LIN {X 0,Y 255.532,Z 417.874,A -85,B 0,C 180,E1 -18352.339,E2 -18352.339} C_VEL
LIN {X 0,Y 254.706,Z 421.868,A -85,B 0,C 180,E1 -18353.296,E2 -18353.296} C_VEL
LIN {X 0,Y 254.484,Z 428.797,A -85,B 0,C 180,E1 -18355.253,E2 -18355.253} C_VEL
LIN {X 0,Y 254.306,Z 433.396,A -85,B 0,C 180,E1 -18356.837,E2 -18356.837} C_VEL
LIN {X 0,Y 254.108,Z 438.832,A -85,B 0,C 180,E1 -18359.213,E2 -18359.213} C_VEL
LIN {X 0,Y 254.235,Z 442.907,A -85,B 0,C 180,E1 -18361.589,E2 -18361.589} C_VEL
LIN {X 0,Y 254.501,Z 444.809,A -85,B 0,C 180,E1 -18363.171,E2 -18363.171} C_VEL
LIN {X 0,Y 254.944,Z 446.181,A -85,B 0,C 180,E1 -18364.749,E2 -18364.749} C_VEL
LIN {X 0,Y 255.447,Z 447.047,A -85,B 0,C 180,E1 -18366.323,E2 -18366.323} C_VEL
LIN {X 0,Y 256.003,Z 447.441,A -85,B 0,C 180,E1 -18367.894,E2 -18367.894} C_VEL
LIN {X 0,Y 256.716,Z 447.298,A -85,B 0,C 180,E1 -18369.459,E2 -18369.459} C_VEL
LIN {X 0,Y 257.985,Z 446.539,A -85,B 0,C 180,E1 -18370.998,E2 -18370.998} C_VEL
LIN {X 0,Y 259.088,Z 445.311,A -85,B 0,C 180,E1 -18372.538,E2 -18372.538} C_VEL
LIN {X 0,Y 261.368,Z 442.495,A -85,B 0,C 180,E1 -18374.805,E2 -18374.805} C_VEL
LIN {X 0,Y 264.023,Z 438.388,A -85,B 0,C 180,E1 -18377.031,E2 -18377.031} C_VEL
LIN {X 0,Y 267.081,Z 432.657,A -85,B 0,C 180,E1 -18379.208,E2 -18379.208} C_VEL
LIN {X 0,Y 270.57,Z 425.346,A -85,B 0,C 180,E1 -18381.329,E2 -18381.329} C_VEL
LIN {X 0,Y 273.754,Z 417.526,A -85,B 0,C 180,E1 -18383.053,E2 -18383.053} C_VEL
LIN {X 0,Y 276.81,Z 408.776,A -85,B 0,C 180,E1 -18384.571,E2 -18384.571} C_VEL
LIN {X 0,Y 280.101,Z 397.834,A -85,B 0,C 180,E1 -18386.05,E2 -18386.05} C_VEL
LIN {X 0,Y 282.427,Z 388.573,A -85,B 0,C 180,E1 -18387.014,E2 -18387.014} C_VEL
LIN {X 0,Y 284.64,Z 377.889,A -85,B 0,C 180,E1 -18387.882,E2 -18387.882} C_VEL
LIN {X 0,Y 286.646,Z 364.758,A -85,B 0,C 180,E1 -18388.634,E2 -18388.634} C_VEL
LIN {X 0,Y 290.224,Z 339.358,A -85,B 0,C 180,E1 -18389.791,E2 -18389.791} C_VEL
LIN {X 0,Y 287.918,Z 334.215,A -85,B 0,C 180,E1 -18391.022,E2 -18391.022} C_VEL
LIN {X 0,Y 285.263,Z 329.062,A -85,B 0,C 180,E1 -18392.583,E2 -18392.583} C_VEL
LIN {X 0,Y 283.342,Z 325.566,A -85,B 0,C 180,E1 -18393.856,E2 -18393.856} C_VEL
LIN {X 0,Y 281.365,Z 322.149,A -85,B 0,C 180,E1 -18395.32,E2 -18395.32} C_VEL
LIN {X 0,Y 278.787,Z 318.232,A -85,B 0,C 180,E1 -18397.663,E2 -18397.663} C_VEL
LIN {X 0,Y 276.577,Z 315.147,A -85,B 0,C 180,E1 -18400.609,E2 -18400.609} C_VEL
LIN {X 0,Y 275.521,Z 314.061,A -85,B 0,C 180,E1 -18403.533,E2 -18403.533} C_VEL
LIN {X 0,Y 275.692,Z 314.436,A -85,B 0,C 180,E1 -18406.695,E2 -18406.695} C_VEL
LIN {X 0,Y 276.651,Z 315.559,A -85,B 0,C 180,E1 -18408.873,E2 -18408.873} C_VEL
LIN {X 0,Y 279.569,Z 320.399,A -85,B 0,C 180,E1 -18412.537,E2 -18412.537} C_VEL
LIN {X 0,Y 282.02,Z 324.321,A -85,B 0,C 180,E1 -18414.58,E2 -18414.58} C_VEL
LIN {X 0,Y 285.054,Z 329.58,A -85,B 0,C 180,E1 -18416.638,E2 -18416.638} C_VEL
LIN {X 0,Y 286.981,Z 333.308,A -85,B 0,C 180,E1 -18417.784,E2 -18417.784} C_VEL
LIN {X 0,Y 287.318,Z 336.449,A -85,B 0,C 180,E1 -18418.229,E2 -18418.229} C_VEL
LIN {X 0,Y 287.621,Z 346.023,A -85,B 0,C 180,E1 -18419.269,E2 -18419.269} C_VEL
LIN {X 0,Y 287.621,Z 359.572,A -85,B 0,C 180,E1 -18420.487,E2 -18420.487} C_VEL
LIN {X 0,Y 285.508,Z 376.187,A -85,B 0,C 180,E1 -18421.308,E2 -18421.308} C_VEL
LIN {X 0,Y 283.222,Z 391.082,A -85,B 0,C 180,E1 -18422.071,E2 -18422.071} C_VEL
LIN {X 0,Y 280.809,Z 401.893,A -85,B 0,C 180,E1 -18422.822,E2 -18422.822} C_VEL
LIN {X 0,Y 277.629,Z 413.56,A -85,B 0,C 180,E1 -18423.906,E2 -18423.906} C_VEL
LIN {X 0,Y 274.246,Z 423.856,A -85,B 0,C 180,E1 -18425.188,E2 -18425.188} C_VEL
LIN {X 0,Y 270.878,Z 433.267,A -85,B 0,C 180,E1 -18426.692,E2 -18426.692} C_VEL
LIN {X 0,Y 267.476,Z 441.522,A -85,B 0,C 180,E1 -18428.416,E2 -18428.416} C_VEL
LIN {X 0,Y 264.494,Z 448.238,A -85,B 0,C 180,E1 -18430.197,E2 -18430.197} C_VEL
LIN {X 0,Y 261.925,Z 453.712,A -85,B 0,C 180,E1 -18432.027,E2 -18432.027} C_VEL
LIN {X 0,Y 259.25,Z 458.894,A -85,B 0,C 180,E1 -18434.271,E2 -18434.271} C_VEL
LIN {X 0,Y 257.239,Z 462.638,A -85,B 0,C 180,E1 -18436.571,E2 -18436.571} C_VEL
LIN {X 0,Y 255.744,Z 465.126,A -85,B 0,C 180,E1 -18438.909,E2 -18438.909} C_VEL
LIN {X 0,Y 255.001,Z 466.213,A -85,B 0,C 180,E1 -18440.481,E2 -18440.481} C_VEL
LIN {X 0,Y 254.485,Z 466.747,A -85,B 0,C 180,E1 -18442.063,E2 -18442.063} C_VEL
LIN {X 0,Y 254.177,Z 466.561,A -85,B 0,C 180,E1 -18444.534,E2 -18444.534} C_VEL
LIN {X 0,Y 254.211,Z 465.734,A -85,B 0,C 180,E1 -18446.433,E2 -18446.433} C_VEL
LIN {X 0,Y 254.165,Z 467.87,A -85,B 0,C 180,E1 -18448.415,E2 -18448.415} C_VEL
LIN {X 0,Y 254.175,Z 468.938,A -85,B 0,C 180,E1 -18450,E2 -18450} C_VEL
LIN {X 0,Y 254.123,Z 469.524,A -85,B 0,C 180,E1 -18451.584,E2 -18451.584} C_VEL
LIN {X 0,Y 254.096,Z 469.648,A -85,B 0,C 180,E1 -18453.171,E2 -18453.171} C_VEL
LIN {X 0,Y 254.098,Z 468.987,A -85,B 0,C 180,E1 -18455.277,E2 -18455.277} C_VEL
LIN {X 0,Y 254.442,Z 466.869,A -85,B 0,C 180,E1 -18457.938,E2 -18457.938} C_VEL
LIN {X 0,Y 255.191,Z 463.773,A -85,B 0,C 180,E1 -18460.312,E2 -18460.312} C_VEL
LIN {X 0,Y 256.366,Z 459.409,A -85,B 0,C 180,E1 -18462.668,E2 -18462.668} C_VEL
LIN {X 0,Y 257.946,Z 453.409,A -85,B 0,C 180,E1 -18465.001,E2 -18465.001} C_VEL
LIN {X 0,Y 259.265,Z 448.471,A -85,B 0,C 180,E1 -18466.536,E2 -18466.536} C_VEL
LIN {X 0,Y 260.845,Z 442.538,A -85,B 0,C 180,E1 -18468.05,E2 -18468.05} C_VEL
LIN {X 0,Y 262.653,Z 435.339,A -85,B 0,C 180,E1 -18469.54,E2 -18469.54} C_VEL
LIN {X 0,Y 264.044,Z 428.911,A -85,B 0,C 180,E1 -18470.651,E2 -18470.651} C_VEL
LIN {X 0,Y 265.617,Z 421.156,A -85,B 0,C 180,E1 -18471.742,E2 -18471.742} C_VEL
LIN {X 0,Y 267.029,Z 413.233,A -85,B 0,C 180,E1 -18472.638,E2 -18472.638} C_VEL
LIN {X 0,Y 268.38,Z 404.327,A -85,B 0,C 180,E1 -18473.419,E2 -18473.419} C_VEL
LIN {X 0,Y 269.583,Z 394.644,A -85,B 0,C 180,E1 -18474.034,E2 -18474.034} C_VEL
LIN {X 0,Y 270.306,Z 385.092,A -85,B 0,C 180,E1 -18474.45,E2 -18474.45} C_VEL
LIN {X 0,Y 271.249,Z 355.127,A -85,B 0,C 180,E1 -18475.292,E2 -18475.292} C_VEL
LIN {X 0,Y 268.624,Z 337.709,A -85,B 0,C 180,E1 -18476.167,E2 -18476.167} C_VEL
LIN {X 0,Y 264.568,Z 317.868,A -85,B 0,C 180,E1 -18477.341,E2 -18477.341} C_VEL
LIN {X 0,Y 262.33,Z 311.832,A -85,B 0,C 180,E1 -18477.854,E2 -18477.854} C_VEL
LIN {X 0,Y 260.483,Z 307.622,A -85,B 0,C 180,E1 -18478.29,E2 -18478.29} C_VEL
LIN {X 0,Y 258.73,Z 299.457,A -85,B 0,C 180,E1 -18481.755,E2 -18481.755} C_VEL
LIN {X 0,Y 256.781,Z 291.051,A -85,B 0,C 180,E1 -18485.563,E2 -18485.563} C_VEL
LIN {X 0,Y 256.133,Z 288.384,A -85,B 0,C 180,E1 -18486.886,E2 -18486.886} C_VEL
LIN {X 0,Y 256.064,Z 288.397,A -85,B 0,C 180,E1 -18491.201,E2 -18491.201} C_VEL
LIN {X 0,Y 256.047,Z 288.404,A -85,B 0,C 180,E1 -18495.532,E2 -18495.532} C_VEL
LIN {X 0,Y 256.018,Z 288.406,A -85,B 0,C 180,E1 -18498.785,E2 -18498.785} C_VEL
LIN {X 0,Y 256.108,Z 288.395,A -85,B 0,C 180,E1 -18502.859,E2 -18502.859} C_VEL
LIN {X 0,Y 256.075,Z 288.398,A -85,B 0,C 180,E1 -18506.704,E2 -18506.704} C_VEL
LIN {X 0,Y 256.064,Z 288.399,A -85,B 0,C 180,E1 -18510.389,E2 -18510.389} C_VEL
LIN {X 0,Y 256.142,Z 288.387,A -85,B 0,C 180,E1 -18514.884,E2 -18514.884} C_VEL
LIN {X 0,Y 256.154,Z 288.377,A -85,B 0,C 180,E1 -18519.099,E2 -18519.099} C_VEL
LIN {X 0,Y 256.264,Z 288.362,A -85,B 0,C 180,E1 -18524.078,E2 -18524.078} C_VEL
LIN {X 0,Y 256.294,Z 288.367,A -85,B 0,C 180,E1 -18527.323,E2 -18527.323} C_VEL
LIN {X 0,Y 256.518,Z 288.339,A -85,B 0,C 180,E1 -18532.122,E2 -18532.122} C_VEL
LIN {X 0,Y 256.487,Z 288.342,A -85,B 0,C 180,E1 -18536.854,E2 -18536.854} C_VEL
LIN {X 0,Y 256.75,Z 288.298,A -85,B 0,C 180,E1 -18539.995,E2 -18539.995} C_VEL
LIN {X 0,Y 256.49,Z 288.343,A -85,B 0,C 180,E1 -18543.136,E2 -18543.136} C_VEL
LIN {X 0,Y 256.492,Z 288.346,A -85,B 0,C 180,E1 -18547.869,E2 -18547.869} C_VEL
LIN {X 0,Y 256.288,Z 288.374,A -85,B 0,C 180,E1 -18552.667,E2 -18552.667} C_VEL
LIN {X 0,Y 256.276,Z 288.365,A -85,B 0,C 180,E1 -18556.297,E2 -18556.297} C_VEL
LIN {X 0,Y 256.148,Z 288.384,A -85,B 0,C 180,E1 -18561.114,E2 -18561.114} C_VEL
LIN {X 0,Y 256.177,Z 288.38,A -85,B 0,C 180,E1 -18565.133,E2 -18565.133} C_VEL
LIN {X 0,Y 256.09,Z 288.397,A -85,B 0,C 180,E1 -18569.596,E2 -18569.596} C_VEL
LIN {X 0,Y 256.052,Z 288.403,A -85,B 0,C 180,E1 -18573.288,E2 -18573.288} C_VEL
LIN {X 0,Y 256.116,Z 288.385,A -85,B 0,C 180,E1 -18577.271,E2 -18577.271} C_VEL
LIN {X 0,Y 256.108,Z 288.387,A -85,B 0,C 180,E1 -18581.184,E2 -18581.184} C_VEL
LIN {X 0,Y 256.148,Z 288.383,A -85,B 0,C 180,E1 -18584.086,E2 -18584.086} C_VEL
LIN {X 0,Y 257.107,Z 291.213,A -85,B 0,C 180,E1 -18584.354,E2 -18584.354} C_VEL
LIN {X 0,Y 258.815,Z 293.87,A -85,B 0,C 180,E1 -18584.707,E2 -18584.707} C_VEL
LIN {X 0,Y 263.773,Z 302.774,A -85,B 0,C 180,E1 -18585.734,E2 -18585.734} C_VEL
LIN {X 0,Y 270.833,Z 318.205,A -85,B 0,C 180,E1 -18587.187,E2 -18587.187} C_VEL
LIN {X 0,Y 272.462,Z 322.528,A -85,B 0,C 180,E1 -18587.532,E2 -18587.532} C_VEL
LIN {X 0,Y 270.884,Z 364.957,A -85,B 0,C 180,E1 -18588.697,E2 -18588.697} C_VEL
LIN {X 0,Y 270.197,Z 375.244,A -85,B 0,C 180,E1 -18589.203,E2 -18589.203} C_VEL
LIN {X 0,Y 268.991,Z 386.83,A -85,B 0,C 180,E1 -18590.078,E2 -18590.078} C_VEL
LIN {X 0,Y 267.757,Z 395.342,A -85,B 0,C 180,E1 -18590.954,E2 -18590.954} C_VEL
LIN {X 0,Y 266.179,Z 404.53,A -85,B 0,C 180,E1 -18592.178,E2 -18592.178} C_VEL
LIN {X 0,Y 264.519,Z 412.588,A -85,B 0,C 180,E1 -18593.525,E2 -18593.525} C_VEL
LIN {X 0,Y 262.892,Z 419.365,A -85,B 0,C 180,E1 -18594.917,E2 -18594.917} C_VEL
LIN {X 0,Y 260.893,Z 427.14,A -85,B 0,C 180,E1 -18596.913,E2 -18596.913} C_VEL
LIN {X 0,Y 259.096,Z 433.249,A -85,B 0,C 180,E1 -18598.978,E2 -18598.978} C_VEL
LIN {X 0,Y 257.954,Z 437.194,A -85,B 0,C 180,E1 -18600.66,E2 -18600.66} C_VEL
LIN {X 0,Y 256.933,Z 440.275,A -85,B 0,C 180,E1 -18602.289,E2 -18602.289} C_VEL
LIN {X 0,Y 256.099,Z 442.685,A -85,B 0,C 180,E1 -18603.955,E2 -18603.955} C_VEL
LIN {X 0,Y 255.374,Z 444.447,A -85,B 0,C 180,E1 -18605.619,E2 -18605.619} C_VEL
LIN {X 0,Y 254.82,Z 445.644,A -85,B 0,C 180,E1 -18607.287,E2 -18607.287} C_VEL
LIN {X 0,Y 254.248,Z 446.491,A -85,B 0,C 180,E1 -18610.004,E2 -18610.004} C_VEL
LIN {X 0,Y 253.968,Z 446.049,A -85,B 0,C 180,E1 -18612.278,E2 -18612.278} C_VEL
LIN {X 0,Y 253.969,Z 445.038,A -85,B 0,C 180,E1 -18613.935,E2 -18613.935} C_VEL
LIN {X 0,Y 254.137,Z 442.565,A -85,B 0,C 180,E1 -18616.405,E2 -18616.405} C_VEL
LIN {X 0,Y 254.518,Z 438.676,A -85,B 0,C 180,E1 -18618.855,E2 -18618.855} C_VEL
LIN {X 0,Y 255.092,Z 433.373,A -85,B 0,C 180,E1 -18621.285,E2 -18621.285} C_VEL
LIN {X 0,Y 255.739,Z 427.604,A -85,B 0,C 180,E1 -18623.318,E2 -18623.318} C_VEL
LIN {X 0,Y 256.559,Z 420.445,A -85,B 0,C 180,E1 -18625.286,E2 -18625.286} C_VEL
LIN {X 0,Y 257.363,Z 413.214,A -85,B 0,C 180,E1 -18626.87,E2 -18626.87} C_VEL
LIN {X 0,Y 258.187,Z 405.508,A -85,B 0,C 180,E1 -18628.245,E2 -18628.245} C_VEL
LIN {X 0,Y 259.028,Z 397.399,A -85,B 0,C 180,E1 -18629.417,E2 -18629.417} C_VEL
LIN {X 0,Y 259.687,Z 389.568,A -85,B 0,C 180,E1 -18630.332,E2 -18630.332} C_VEL
LIN {X 0,Y 260.272,Z 380.968,A -85,B 0,C 180,E1 -18631.124,E2 -18631.124} C_VEL
LIN {X 0,Y 260.767,Z 370.639,A -85,B 0,C 180,E1 -18631.822,E2 -18631.822} C_VEL
LIN {X 0,Y 261.173,Z 358.837,A -85,B 0,C 180,E1 -18632.318,E2 -18632.318} C_VEL
LIN {X 0,Y 262.088,Z 311.721,A -85,B 0,C 180,E1 -18633.604,E2 -18633.604} C_VEL
LIN {X 0,Y 260.06,Z 299.467,A -85,B 0,C 180,E1 -18634.081,E2 -18634.081} C_VEL
LIN {X 0,Y 256.313,Z 288.374,A -85,B 0,C 180,E1 -18634.661,E2 -18634.661} C_VEL
LIN {X 0,Y 256.483,Z 288.346,A -85,B 0,C 180,E1 -18637.875,E2 -18637.875} C_VEL
LIN {X 0,Y 256.23,Z 288.376,A -85,B 0,C 180,E1 -18642.676,E2 -18642.676} C_VEL
LIN {X 0,Y 256.218,Z 288.379,A -85,B 0,C 180,E1 -18646.277,E2 -18646.277} C_VEL
LIN {X 0,Y 256.135,Z 288.391,A -85,B 0,C 180,E1 -18650.898,E2 -18650.898} C_VEL
LIN {X 0,Y 256.105,Z 288.396,A -85,B 0,C 180,E1 -18655.115,E2 -18655.115} C_VEL
LIN {X 0,Y 256.025,Z 288.404,A -85,B 0,C 180,E1 -18659.611,E2 -18659.611} C_VEL
LIN {X 0,Y 256.041,Z 288.4,A -85,B 0,C 180,E1 -18663.297,E2 -18663.297} C_VEL
LIN {X 0,Y 256.093,Z 288.396,A -85,B 0,C 180,E1 -18667.275,E2 -18667.275} C_VEL
LIN {X 0,Y 256.036,Z 288.402,A -85,B 0,C 180,E1 -18672.182,E2 -18672.182} C_VEL
LIN {X 0,Y 256.03,Z 288.403,A -85,B 0,C 180,E1 -18676.675,E2 -18676.675} C_VEL
LIN {X 0,Y 256.055,Z 288.397,A -85,B 0,C 180,E1 -18680.863,E2 -18680.863} C_VEL
LIN {X 0,Y 256.116,Z 288.392,A -85,B 0,C 180,E1 -18682.873,E2 -18682.873} C_VEL
LIN {X 0,Y 256.052,Z 288.398,A -85,B 0,C 180,E1 -18686.712,E2 -18686.712} C_VEL
LIN {X 0,Y 256.043,Z 288.402,A -85,B 0,C 180,E1 -18690.398,E2 -18690.398} C_VEL
LIN {X 0,Y 256.124,Z 288.388,A -85,B 0,C 180,E1 -18694.894,E2 -18694.894} C_VEL
LIN {X 0,Y 256.154,Z 288.375,A -85,B 0,C 180,E1 -18699.11,E2 -18699.11} C_VEL
LIN {X 0,Y 256.386,Z 288.337,A -85,B 0,C 180,E1 -18702.147,E2 -18702.147} C_VEL
LIN {X 0,Y 258.584,Z 308.952,A -85,B 0,C 180,E1 -18703.136,E2 -18703.136} C_VEL
LIN {X 0,Y 257.215,Z 365.235,A -85,B 0,C 180,E1 -18705.72,E2 -18705.72} C_VEL
LIN {X 0,Y 256.873,Z 376.015,A -85,B 0,C 180,E1 -18706.457,E2 -18706.457} C_VEL
LIN {X 0,Y 256.429,Z 387.695,A -85,B 0,C 180,E1 -18707.541,E2 -18707.541} C_VEL
LIN {X 0,Y 255.881,Z 398.365,A -85,B 0,C 180,E1 -18708.881,E2 -18708.881} C_VEL
LIN {X 0,Y 255.407,Z 407.479,A -85,B 0,C 180,E1 -18710.303,E2 -18710.303} C_VEL
LIN {X 0,Y 254.959,Z 416.652,A -85,B 0,C 180,E1 -18712.083,E2 -18712.083} C_VEL
LIN {X 0,Y 254.706,Z 421.868,A -85,B 0,C 180,E1 -18713.296,E2 -18713.296} C_VEL
LIN {X 0,Y 253.879,Z 425.701,A -85,B 0,C 180,E1 -18714.293,E2 -18714.293} C_VEL
LIN {X 0,Y 252.144,Z 429.067,A -85,B 0,C 180,E1 -18715.334,E2 -18715.334} C_VEL
LIN {X 0,Y 247.736,Z 435.645,A -85,B 0,C 180,E1 -18717.981,E2 -18717.981} C_VEL
LIN {X 0,Y 247.036,Z 438.202,A -85,B 0,C 180,E1 -18719.221,E2 -18719.221} C_VEL
LIN {X 0,Y 247.165,Z 442.474,A -85,B 0,C 180,E1 -18721.635,E2 -18721.635} C_VEL
LIN {X 0,Y 247.44,Z 444.59,A -85,B 0,C 180,E1 -18723.262,E2 -18723.262} C_VEL
LIN {X 0,Y 247.875,Z 446.181,A -85,B 0,C 180,E1 -18724.884,E2 -18724.884} C_VEL
LIN {X 0,Y 248.399,Z 447.279,A -85,B 0,C 180,E1 -18726.503,E2 -18726.503} C_VEL
LIN {X 0,Y 248.99,Z 447.808,A -85,B 0,C 180,E1 -18728.118,E2 -18728.118} C_VEL
LIN {X 0,Y 249.748,Z 447.791,A -85,B 0,C 180,E1 -18729.725,E2 -18729.725} C_VEL
LIN {X 0,Y 251.982,Z 446.617,A -85,B 0,C 180,E1 -18732.529,E2 -18732.529} C_VEL
LIN {X 0,Y 253.831,Z 444.809,A -85,B 0,C 180,E1 -18734.434,E2 -18734.434} C_VEL
LIN {X 0,Y 256.432,Z 441.402,A -85,B 0,C 180,E1 -18736.729,E2 -18736.729} C_VEL
LIN {X 0,Y 259.51,Z 436.674,A -85,B 0,C 180,E1 -18738.969,E2 -18738.969} C_VEL
LIN {X 0,Y 262.426,Z 431.601,A -85,B 0,C 180,E1 -18740.789,E2 -18740.789} C_VEL
LIN {X 0,Y 266.277,Z 423.768,A -85,B 0,C 180,E1 -18742.916,E2 -18742.916} C_VEL
LIN {X 0,Y 269.7,Z 415.546,A -85,B 0,C 180,E1 -18744.646,E2 -18744.646} C_VEL
LIN {X 0,Y 273.107,Z 406.397,A -85,B 0,C 180,E1 -18746.152,E2 -18746.152} C_VEL
LIN {X 0,Y 275.839,Z 397.449,A -85,B 0,C 180,E1 -18747.302,E2 -18747.302} C_VEL
LIN {X 0,Y 278.735,Z 386.349,A -85,B 0,C 180,E1 -18748.423,E2 -18748.423} C_VEL
LIN {X 0,Y 281.214,Z 374.18,A -85,B 0,C 180,E1 -18749.324,E2 -18749.324} C_VEL
LIN {X 0,Y 283.64,Z 358.651,A -85,B 0,C 180,E1 -18750.105,E2 -18750.105} C_VEL
LIN {X 0,Y 285.914,Z 342.529,A -85,B 0,C 180,E1 -18750.895,E2 -18750.895} C_VEL
LIN {X 0,Y 282.76,Z 335.677,A -85,B 0,C 180,E1 -18752.844,E2 -18752.844} C_VEL
LIN {X 0,Y 280.376,Z 331.231,A -85,B 0,C 180,E1 -18754.527,E2 -18754.527} C_VEL
LIN {X 0,Y 278.688,Z 328.177,A -85,B 0,C 180,E1 -18755.937,E2 -18755.937} C_VEL
LIN {X 0,Y 276.709,Z 324.937,A -85,B 0,C 180,E1 -18757.898,E2 -18757.898} C_VEL
LIN {X 0,Y 274.619,Z 321.903,A -85,B 0,C 180,E1 -18760.838,E2 -18760.838} C_VEL
LIN {X 0,Y 273.818,Z 320.976,A -85,B 0,C 180,E1 -18763.003,E2 -18763.003} C_VEL
LIN {X 0,Y 273.879,Z 321.279,A -85,B 0,C 180,E1 -18766.582,E2 -18766.582} C_VEL
LIN {X 0,Y 274.736,Z 322.335,A -85,B 0,C 180,E1 -18768.663,E2 -18768.663} C_VEL
LIN {X 0,Y 277.302,Z 326.87,A -85,B 0,C 180,E1 -18772.161,E2 -18772.161} C_VEL
LIN {X 0,Y 279.521,Z 330.618,A -85,B 0,C 180,E1 -18774.154,E2 -18774.154} C_VEL
LIN {X 0,Y 282.209,Z 335.555,A -85,B 0,C 180,E1 -18776.125,E2 -18776.125} C_VEL
LIN {X 0,Y 283.577,Z 338.512,A -85,B 0,C 180,E1 -18777.064,E2 -18777.064} C_VEL
LIN {X 0,Y 283.745,Z 348.629,A -85,B 0,C 180,E1 -18778.198,E2 -18778.198} C_VEL
LIN {X 0,Y 283.486,Z 361.625,A -85,B 0,C 180,E1 -18779.407,E2 -18779.407} C_VEL
LIN {X 0,Y 279.505,Z 388.455,A -85,B 0,C 180,E1 -18780.742,E2 -18780.742} C_VEL
LIN {X 0,Y 276.722,Z 400.474,A -85,B 0,C 180,E1 -18781.562,E2 -18781.562} C_VEL
LIN {X 0,Y 273.346,Z 412.373,A -85,B 0,C 180,E1 -18782.639,E2 -18782.639} C_VEL
LIN {X 0,Y 269.76,Z 422.749,A -85,B 0,C 180,E1 -18783.919,E2 -18783.919} C_VEL
LIN {X 0,Y 266.857,Z 430.22,A -85,B 0,C 180,E1 -18785.078,E2 -18785.078} C_VEL
LIN {X 0,Y 263.126,Z 439.07,A -85,B 0,C 180,E1 -18786.798,E2 -18786.798} C_VEL
LIN {X 0,Y 259.76,Z 446.155,A -85,B 0,C 180,E1 -18788.577,E2 -18788.577} C_VEL
LIN {X 0,Y 257.379,Z 450.864,A -85,B 0,C 180,E1 -18790.042,E2 -18790.042} C_VEL
LIN {X 0,Y 254.317,Z 456.485,A -85,B 0,C 180,E1 -18792.303,E2 -18792.303} C_VEL
LIN {X 0,Y 251.72,Z 460.782,A -85,B 0,C 180,E1 -18794.618,E2 -18794.618} C_VEL
LIN {X 0,Y 249.752,Z 463.822,A -85,B 0,C 180,E1 -18796.99,E2 -18796.99} C_VEL
LIN {X 0,Y 248.765,Z 465.133,A -85,B 0,C 180,E1 -18798.594,E2 -18798.594} C_VEL
LIN {X 0,Y 247.987,Z 465.972,A -85,B 0,C 180,E1 -18800.209,E2 -18800.209} C_VEL
LIN {X 0,Y 247.442,Z 466.357,A -85,B 0,C 180,E1 -18801.835,E2 -18801.835} C_VEL
LIN {X 0,Y 247.184,Z 466.23,A -85,B 0,C 180,E1 -18803.469,E2 -18803.469} C_VEL
LIN {X 0,Y 247.164,Z 464.91,A -85,B 0,C 180,E1 -18806.127,E2 -18806.127} C_VEL
LIN {X 0,Y 247.093,Z 467.393,A -85,B 0,C 180,E1 -18808.37,E2 -18808.37} C_VEL
LIN {X 0,Y 247.099,Z 468.522,A -85,B 0,C 180,E1 -18810,E2 -18810} C_VEL
LIN {X 0,Y 247.051,Z 469.167,A -85,B 0,C 180,E1 -18811.63,E2 -18811.63} C_VEL
LIN {X 0,Y 247.011,Z 469.349,A -85,B 0,C 180,E1 -18813.262,E2 -18813.262} C_VEL
LIN {X 0,Y 247.003,Z 468.88,A -85,B 0,C 180,E1 -18815.181,E2 -18815.181} C_VEL
LIN {X 0,Y 247.402,Z 466.688,A -85,B 0,C 180,E1 -18818.165,E2 -18818.165} C_VEL
LIN {X 0,Y 248.205,Z 463.655,A -85,B 0,C 180,E1 -18820.605,E2 -18820.605} C_VEL
LIN {X 0,Y 249.434,Z 459.378,A -85,B 0,C 180,E1 -18823.026,E2 -18823.026} C_VEL
LIN {X 0,Y 251.104,Z 453.525,A -85,B 0,C 180,E1 -18825.42,E2 -18825.42} C_VEL
LIN {X 0,Y 252.882,Z 447.267,A -85,B 0,C 180,E1 -18827.383,E2 -18827.383} C_VEL
LIN {X 0,Y 254.604,Z 441.165,A -85,B 0,C 180,E1 -18828.925,E2 -18828.925} C_VEL
LIN {X 0,Y 256.237,Z 434.785,A -85,B 0,C 180,E1 -18830.259,E2 -18830.259} C_VEL
LIN {X 0,Y 257.437,Z 429.537,A -85,B 0,C 180,E1 -18831.206,E2 -18831.206} C_VEL
LIN {X 0,Y 259.353,Z 420.498,A -85,B 0,C 180,E1 -18832.505,E2 -18832.505} C_VEL
LIN {X 0,Y 260.848,Z 412.492,A -85,B 0,C 180,E1 -18833.416,E2 -18833.416} C_VEL
LIN {X 0,Y 262.142,Z 404.259,A -85,B 0,C 180,E1 -18834.152,E2 -18834.152} C_VEL
LIN {X 0,Y 263.414,Z 394.577,A -85,B 0,C 180,E1 -18834.78,E2 -18834.78} C_VEL
LIN {X 0,Y 264.136,Z 385.446,A -85,B 0,C 180,E1 -18835.196,E2 -18835.196} C_VEL
LIN {X 0,Y 265.131,Z 356.256,A -85,B 0,C 180,E1 -18836.038,E2 -18836.038} C_VEL
LIN {X 0,Y 263.066,Z 341.866,A -85,B 0,C 180,E1 -18836.774,E2 -18836.774} C_VEL
LIN {X 0,Y 259.448,Z 323.133,A -85,B 0,C 180,E1 -18837.895,E2 -18837.895} C_VEL
LIN {X 0,Y 258.175,Z 318.358,A -85,B 0,C 180,E1 -18838.242,E2 -18838.242} C_VEL
LIN {X 0,Y 254.158,Z 309.74,A -85,B 0,C 180,E1 -18839.145,E2 -18839.145} C_VEL
LIN {X 0,Y 253.208,Z 307.156,A -85,B 0,C 180,E1 -18839.43,E2 -18839.43} C_VEL
LIN {X 0,Y 251.27,Z 298.315,A -85,B 0,C 180,E1 -18843.373,E2 -18843.373} C_VEL
LIN {X 0,Y 249.61,Z 291.26,A -85,B 0,C 180,E1 -18846.749,E2 -18846.749} C_VEL
LIN {X 0,Y 249.043,Z 289.279,A -85,B 0,C 180,E1 -18847.794,E2 -18847.794} C_VEL
LIN {X 0,Y 249.017,Z 289.279,A -85,B 0,C 180,E1 -18850.476,E2 -18850.476} C_VEL
LIN {X 0,Y 248.993,Z 289.277,A -85,B 0,C 180,E1 -18854.881,E2 -18854.881} C_VEL
LIN {X 0,Y 248.993,Z 289.276,A -85,B 0,C 180,E1 -18857.353,E2 -18857.353} C_VEL
LIN {X 0,Y 249.048,Z 289.273,A -85,B 0,C 180,E1 -18862.199,E2 -18862.199} C_VEL
LIN {X 0,Y 249.052,Z 289.267,A -85,B 0,C 180,E1 -18865.636,E2 -18865.636} C_VEL
LIN {X 0,Y 249.011,Z 289.269,A -85,B 0,C 180,E1 -18869.463,E2 -18869.463} C_VEL
LIN {X 0,Y 249.045,Z 289.266,A -85,B 0,C 180,E1 -18873.154,E2 -18873.154} C_VEL
LIN {X 0,Y 249.063,Z 289.272,A -85,B 0,C 180,E1 -18876.726,E2 -18876.726} C_VEL
LIN {X 0,Y 249.096,Z 289.265,A -85,B 0,C 180,E1 -18880.206,E2 -18880.206} C_VEL
LIN {X 0,Y 249.201,Z 289.242,A -85,B 0,C 180,E1 -18883.614,E2 -18883.614} C_VEL
LIN {X 0,Y 249.247,Z 289.232,A -85,B 0,C 180,E1 -18888.611,E2 -18888.611} C_VEL
LIN {X 0,Y 249.458,Z 289.22,A -85,B 0,C 180,E1 -18891.897,E2 -18891.897} C_VEL
LIN {X 0,Y 249.285,Z 289.229,A -85,B 0,C 180,E1 -18895.143,E2 -18895.143} C_VEL
LIN {X 0,Y 249.672,Z 289.187,A -85,B 0,C 180,E1 -18898.382,E2 -18898.382} C_VEL
LIN {X 0,Y 249.672,Z 289.188,A -85,B 0,C 180,E1 -18901.608,E2 -18901.608} C_VEL
LIN {X 0,Y 249.427,Z 289.217,A -85,B 0,C 180,E1 -18906.58,E2 -18906.58} C_VEL
LIN {X 0,Y 249.339,Z 289.229,A -85,B 0,C 180,E1 -18909.731,E2 -18909.731} C_VEL
LIN {X 0,Y 249.199,Z 289.249,A -85,B 0,C 180,E1 -18914.698,E2 -18914.698} C_VEL
LIN {X 0,Y 249.132,Z 289.265,A -85,B 0,C 180,E1 -18918.072,E2 -18918.072} C_VEL
LIN {X 0,Y 249.078,Z 289.267,A -85,B 0,C 180,E1 -18921.513,E2 -18921.513} C_VEL
LIN {X 0,Y 249.119,Z 289.262,A -85,B 0,C 180,E1 -18925.477,E2 -18925.477} C_VEL
LIN {X 0,Y 249.06,Z 289.269,A -85,B 0,C 180,E1 -18928.984,E2 -18928.984} C_VEL
LIN {X 0,Y 249.015,Z 289.276,A -85,B 0,C 180,E1 -18932.421,E2 -18932.421} C_VEL
LIN {X 0,Y 249.043,Z 289.258,A -85,B 0,C 180,E1 -18936.335,E2 -18936.335} C_VEL
LIN {X 0,Y 249.064,Z 289.261,A -85,B 0,C 180,E1 -18940.458,E2 -18940.458} C_VEL
LIN {X 0,Y 249.073,Z 289.27,A -85,B 0,C 180,E1 -18942.986,E2 -18942.986} C_VEL
LIN {X 0,Y 250.053,Z 292.07,A -85,B 0,C 180,E1 -18943.253,E2 -18943.253} C_VEL
LIN {X 0,Y 251.663,Z 294.475,A -85,B 0,C 180,E1 -18943.602,E2 -18943.602} C_VEL
LIN {X 0,Y 257.999,Z 305.545,A -85,B 0,C 180,E1 -18944.976,E2 -18944.976} C_VEL
LIN {X 0,Y 263.869,Z 318.195,A -85,B 0,C 180,E1 -18946.249,E2 -18946.249} C_VEL
LIN {X 0,Y 266.364,Z 324.215,A -85,B 0,C 180,E1 -18946.783,E2 -18946.783} C_VEL
LIN {X 0,Y 264.785,Z 365.07,A -85,B 0,C 180,E1 -18947.927,E2 -18947.927} C_VEL
LIN {X 0,Y 264.146,Z 374.652,A -85,B 0,C 180,E1 -18948.401,E2 -18948.401} C_VEL
LIN {X 0,Y 262.965,Z 385.914,A -85,B 0,C 180,E1 -18949.223,E2 -18949.223} C_VEL
LIN {X 0,Y 261.374,Z 396.3,A -85,B 0,C 180,E1 -18950.312,E2 -18950.312} C_VEL
LIN {X 0,Y 260.044,Z 403.809,A -85,B 0,C 180,E1 -18951.32,E2 -18951.32} C_VEL
LIN {X 0,Y 258.647,Z 410.534,A -85,B 0,C 180,E1 -18952.408,E2 -18952.408} C_VEL
LIN {X 0,Y 256.765,Z 418.256,A -85,B 0,C 180,E1 -18953.951,E2 -18953.951} C_VEL
LIN {X 0,Y 255.192,Z 424.21,A -85,B 0,C 180,E1 -18955.412,E2 -18955.412} C_VEL
LIN {X 0,Y 253.78,Z 429.083,A -85,B 0,C 180,E1 -18956.843,E2 -18956.843} C_VEL
LIN {X 0,Y 252.314,Z 433.775,A -85,B 0,C 180,E1 -18958.516,E2 -18958.516} C_VEL
LIN {X 0,Y 251.154,Z 437.513,A -85,B 0,C 180,E1 -18960.151,E2 -18960.151} C_VEL
LIN {X 0,Y 249.802,Z 441.336,A -85,B 0,C 180,E1 -18962.341,E2 -18962.341} C_VEL
LIN {X 0,Y 248.582,Z 444.438,A -85,B 0,C 180,E1 -18964.907,E2 -18964.907} C_VEL
LIN {X 0,Y 247.918,Z 445.776,A -85,B 0,C 180,E1 -18966.617,E2 -18966.617} C_VEL
LIN {X 0,Y 247.465,Z 446.573,A -85,B 0,C 180,E1 -18968.334,E2 -18968.334} C_VEL
LIN {X 0,Y 247.153,Z 446.834,A -85,B 0,C 180,E1 -18970.048,E2 -18970.048} C_VEL
LIN {X 0,Y 246.929,Z 446.483,A -85,B 0,C 180,E1 -18971.755,E2 -18971.755} C_VEL
LIN {X 0,Y 246.855,Z 445.582,A -85,B 0,C 180,E1 -18973.459,E2 -18973.459} C_VEL
LIN {X 0,Y 246.929,Z 443.947,A -85,B 0,C 180,E1 -18975.368,E2 -18975.368} C_VEL
LIN {X 0,Y 247.236,Z 440.989,A -85,B 0,C 180,E1 -18977.691,E2 -18977.691} C_VEL
LIN {X 0,Y 247.725,Z 436.459,A -85,B 0,C 180,E1 -18980.2,E2 -18980.2} C_VEL
LIN {X 0,Y 248.28,Z 431.771,A -85,B 0,C 180,E1 -18982.141,E2 -18982.141} C_VEL
LIN {X 0,Y 248.792,Z 426.457,A -85,B 0,C 180,E1 -18983.919,E2 -18983.919} C_VEL
LIN {X 0,Y 249.554,Z 420.461,A -85,B 0,C 180,E1 -18985.559,E2 -18985.559} C_VEL
LIN {X 0,Y 250.394,Z 413.168,A -85,B 0,C 180,E1 -18987.185,E2 -18987.185} C_VEL
LIN {X 0,Y 251.27,Z 405.38,A -85,B 0,C 180,E1 -18988.598,E2 -18988.598} C_VEL
LIN {X 0,Y 252.126,Z 397.179,A -85,B 0,C 180,E1 -18989.801,E2 -18989.801} C_VEL
LIN {X 0,Y 252.8,Z 389.539,A -85,B 0,C 180,E1 -18990.705,E2 -18990.705} C_VEL
LIN {X 0,Y 253.455,Z 379.956,A -85,B 0,C 180,E1 -18991.589,E2 -18991.589} C_VEL
LIN {X 0,Y 254.001,Z 369.105,A -85,B 0,C 180,E1 -18992.306,E2 -18992.306} C_VEL
LIN {X 0,Y 254.389,Z 354.396,A -85,B 0,C 180,E1 -18992.841,E2 -18992.841} C_VEL
LIN {X 0,Y 255.313,Z 312.699,A -85,B 0,C 180,E1 -18994.001,E2 -18994.001} C_VEL
LIN {X 0,Y 253.275,Z 300.812,A -85,B 0,C 180,E1 -18994.485,E2 -18994.485} C_VEL
LIN {X 0,Y 249.307,Z 289.354,A -85,B 0,C 180,E1 -18995.099,E2 -18995.099} C_VEL
LIN {X 0,Y 249.423,Z 289.225,A -85,B 0,C 180,E1 -18998.099,E2 -18998.099} C_VEL
LIN {X 0,Y 249.163,Z 289.258,A -85,B 0,C 180,E1 -19003.042,E2 -19003.042} C_VEL
LIN {X 0,Y 249.166,Z 289.257,A -85,B 0,C 180,E1 -19006.488,E2 -19006.488} C_VEL
LIN {X 0,Y 249.066,Z 289.276,A -85,B 0,C 180,E1 -19011.401,E2 -19011.401} C_VEL
LIN {X 0,Y 249.058,Z 289.275,A -85,B 0,C 180,E1 -19015.463,E2 -19015.463} C_VEL
LIN {X 0,Y 249.008,Z 289.279,A -85,B 0,C 180,E1 -19018.976,E2 -19018.976} C_VEL
LIN {X 0,Y 249.002,Z 289.274,A -85,B 0,C 180,E1 -19022.43,E2 -19022.43} C_VEL
LIN {X 0,Y 248.989,Z 289.279,A -85,B 0,C 180,E1 -19026.353,E2 -19026.353} C_VEL
LIN {X 0,Y 248.962,Z 289.283,A -85,B 0,C 180,E1 -19030.487,E2 -19030.487} C_VEL
LIN {X 0,Y 248.963,Z 289.281,A -85,B 0,C 180,E1 -19034.889,E2 -19034.889} C_VEL
LIN {X 0,Y 248.991,Z 289.281,A -85,B 0,C 180,E1 -19037.366,E2 -19037.366} C_VEL
LIN {X 0,Y 249.01,Z 289.278,A -85,B 0,C 180,E1 -19041.625,E2 -19041.625} C_VEL
LIN {X 0,Y 249.03,Z 289.278,A -85,B 0,C 180,E1 -19045.645,E2 -19045.645} C_VEL
LIN {X 0,Y 248.99,Z 289.28,A -85,B 0,C 180,E1 -19049.472,E2 -19049.472} C_VEL
LIN {X 0,Y 249.025,Z 289.275,A -85,B 0,C 180,E1 -19053.164,E2 -19053.164} C_VEL
LIN {X 0,Y 249.047,Z 289.265,A -85,B 0,C 180,E1 -19056.736,E2 -19056.736} C_VEL
LIN {X 0,Y 249.345,Z 289.214,A -85,B 0,C 180,E1 -19062.131,E2 -19062.131} C_VEL
LIN {X 0,Y 251.494,Z 310.031,A -85,B 0,C 180,E1 -19063.145,E2 -19063.145} C_VEL
LIN {X 0,Y 250.111,Z 365.964,A -85,B 0,C 180,E1 -19065.824,E2 -19065.824} C_VEL
LIN {X 0,Y 249.729,Z 376.583,A -85,B 0,C 180,E1 -19066.581,E2 -19066.581} C_VEL
LIN {X 0,Y 249.369,Z 387.298,A -85,B 0,C 180,E1 -19067.596,E2 -19067.596} C_VEL
LIN {X 0,Y 248.785,Z 398.415,A -85,B 0,C 180,E1 -19069.013,E2 -19069.013} C_VEL
LIN {X 0,Y 248.326,Z 407.345,A -85,B 0,C 180,E1 -19070.435,E2 -19070.435} C_VEL
LIN {X 0,Y 247.874,Z 416.601,A -85,B 0,C 180,E1 -19072.266,E2 -19072.266} C_VEL
LIN {X 0,Y 247.525,Z 423.237,A -85,B 0,C 180,E1 -19073.903,E2 -19073.903} C_VEL
LIN {X 0,Y 247.409,Z 429.995,A -85,B 0,C 180,E1 -19075.933,E2 -19075.933} C_VEL
LIN {X 0,Y 247.104,Z 435.434,A -85,B 0,C 180,E1 -19077.968,E2 -19077.968} C_VEL
LIN {X 0,Y 247.036,Z 438.202,A -85,B 0,C 180,E1 -19079.221,E2 -19079.221} C_VEL
LIN {X 0,Y 246.403,Z 440.606,A -85,B 0,C 180,E1 -19080.475,E2 -19080.475} C_VEL
LIN {X 0,Y 243.774,Z 443.625,A -85,B 0,C 180,E1 -19082.592,E2 -19082.592} C_VEL
LIN {X 0,Y 241.73,Z 445.491,A -85,B 0,C 180,E1 -19084.357,E2 -19084.357} C_VEL
LIN {X 0,Y 241.095,Z 446.672,A -85,B 0,C 180,E1 -19085.732,E2 -19085.732} C_VEL
LIN {X 0,Y 241.171,Z 446.982,A -85,B 0,C 180,E1 -19086.195,E2 -19086.195} C_VEL
LIN {X 0,Y 241.964,Z 448.044,A -85,B 0,C 180,E1 -19088.356,E2 -19088.356} C_VEL
LIN {X 0,Y 242.776,Z 448.285,A -85,B 0,C 180,E1 -19090.008,E2 -19090.008} C_VEL
LIN {X 0,Y 244.143,Z 448.032,A -85,B 0,C 180,E1 -19091.63,E2 -19091.63} C_VEL
LIN {X 0,Y 245.387,Z 447.256,A -85,B 0,C 180,E1 -19093.25,E2 -19093.25} C_VEL
LIN {X 0,Y 247.046,Z 445.874,A -85,B 0,C 180,E1 -19094.84,E2 -19094.84} C_VEL
LIN {X 0,Y 249.802,Z 442.956,A -85,B 0,C 180,E1 -19097.187,E2 -19097.187} C_VEL
LIN {X 0,Y 253.046,Z 438.615,A -85,B 0,C 180,E1 -19099.473,E2 -19099.473} C_VEL
LIN {X 0,Y 256.052,Z 433.86,A -85,B 0,C 180,E1 -19101.331,E2 -19101.331} C_VEL
LIN {X 0,Y 259.38,Z 427.992,A -85,B 0,C 180,E1 -19103.139,E2 -19103.139} C_VEL
LIN {X 0,Y 262.98,Z 420.779,A -85,B 0,C 180,E1 -19104.897,E2 -19104.897} C_VEL
LIN {X 0,Y 266.815,Z 411.613,A -85,B 0,C 180,E1 -19106.606,E2 -19106.606} C_VEL
LIN {X 0,Y 270.099,Z 402.671,A -85,B 0,C 180,E1 -19107.932,E2 -19107.932} C_VEL
LIN {X 0,Y 273.568,Z 391.333,A -85,B 0,C 180,E1 -19109.221,E2 -19109.221} C_VEL
LIN {X 0,Y 276.014,Z 381.224,A -85,B 0,C 180,E1 -19110.09,E2 -19110.09} C_VEL
LIN {X 0,Y 278.297,Z 369.687,A -85,B 0,C 180,E1 -19110.829,E2 -19110.829} C_VEL
LIN {X 0,Y 281.944,Z 346.313,A -85,B 0,C 180,E1 -19111.977,E2 -19111.977} C_VEL
LIN {X 0,Y 279.589,Z 341.037,A -85,B 0,C 180,E1 -19113.61,E2 -19113.61} C_VEL
LIN {X 0,Y 277.823,Z 337.512,A -85,B 0,C 180,E1 -19114.961,E2 -19114.961} C_VEL
LIN {X 0,Y 276.141,Z 334.34,A -85,B 0,C 180,E1 -19116.468,E2 -19116.468} C_VEL
LIN {X 0,Y 274.49,Z 331.478,A -85,B 0,C 180,E1 -19118.277,E2 -19118.277} C_VEL
LIN {X 0,Y 272.658,Z 328.588,A -85,B 0,C 180,E1 -19121.209,E2 -19121.209} C_VEL
LIN {X 0,Y 271.925,Z 327.798,A -85,B 0,C 180,E1 -19123.641,E2 -19123.641} C_VEL
LIN {X 0,Y 272.215,Z 328.277,A -85,B 0,C 180,E1 -19127.072,E2 -19127.072} C_VEL
LIN {X 0,Y 272.865,Z 329.27,A -85,B 0,C 180,E1 -19128.591,E2 -19128.591} C_VEL
LIN {X 0,Y 275.214,Z 333.651,A -85,B 0,C 180,E1 -19131.969,E2 -19131.969} C_VEL
LIN {X 0,Y 277.012,Z 336.938,A -85,B 0,C 180,E1 -19133.719,E2 -19133.719} C_VEL
LIN {X 0,Y 279.476,Z 341.763,A -85,B 0,C 180,E1 -19135.68,E2 -19135.68} C_VEL
LIN {X 0,Y 280.154,Z 343.254,A -85,B 0,C 180,E1 -19136.168,E2 -19136.168} C_VEL
LIN {X 0,Y 279.997,Z 352.566,A -85,B 0,C 180,E1 -19137.227,E2 -19137.227} C_VEL
LIN {X 0,Y 279.599,Z 363.72,A -85,B 0,C 180,E1 -19138.268,E2 -19138.268} C_VEL
LIN {X 0,Y 275.744,Z 387.327,A -85,B 0,C 180,E1 -19139.459,E2 -19139.459} C_VEL
LIN {X 0,Y 272.823,Z 399.55,A -85,B 0,C 180,E1 -19140.272,E2 -19140.272} C_VEL
LIN {X 0,Y 269.778,Z 409.853,A -85,B 0,C 180,E1 -19141.187,E2 -19141.187} C_VEL
LIN {X 0,Y 265.883,Z 420.689,A -85,B 0,C 180,E1 -19142.446,E2 -19142.446} C_VEL
LIN {X 0,Y 262.364,Z 429.31,A -85,B 0,C 180,E1 -19143.769,E2 -19143.769} C_VEL
LIN {X 0,Y 259.059,Z 436.575,A -85,B 0,C 180,E1 -19145.134,E2 -19145.134} C_VEL
LIN {X 0,Y 255.354,Z 444.058,A -85,B 0,C 180,E1 -19146.908,E2 -19146.908} C_VEL
LIN {X 0,Y 251.416,Z 451.117,A -85,B 0,C 180,E1 -19149.12,E2 -19149.12} C_VEL
LIN {X 0,Y 248.625,Z 455.786,A -85,B 0,C 180,E1 -19151.029,E2 -19151.029} C_VEL
LIN {X 0,Y 245.663,Z 460.104,A -85,B 0,C 180,E1 -19153.376,E2 -19153.376} C_VEL
LIN {X 0,Y 244.158,Z 462.279,A -85,B 0,C 180,E1 -19154.985,E2 -19154.985} C_VEL
LIN {X 0,Y 242.841,Z 463.97,A -85,B 0,C 180,E1 -19156.613,E2 -19156.613} C_VEL
LIN {X 0,Y 241.802,Z 465.144,A -85,B 0,C 180,E1 -19158.261,E2 -19158.261} C_VEL
LIN {X 0,Y 240.989,Z 465.738,A -85,B 0,C 180,E1 -19159.922,E2 -19159.922} C_VEL
LIN {X 0,Y 240.418,Z 465.868,A -85,B 0,C 180,E1 -19161.595,E2 -19161.595} C_VEL
LIN {X 0,Y 240.107,Z 465.044,A -85,B 0,C 180,E1 -19164.412,E2 -19164.412} C_VEL
LIN {X 0,Y 240.133,Z 464.136,A -85,B 0,C 180,E1 -19165.85,E2 -19165.85} C_VEL
LIN {X 0,Y 240.023,Z 466.917,A -85,B 0,C 180,E1 -19168.322,E2 -19168.322} C_VEL
LIN {X 0,Y 240.025,Z 468.105,A -85,B 0,C 180,E1 -19170,E2 -19170} C_VEL
LIN {X 0,Y 239.979,Z 468.809,A -85,B 0,C 180,E1 -19171.678,E2 -19171.678} C_VEL
LIN {X 0,Y 239.927,Z 469.039,A -85,B 0,C 180,E1 -19173.358,E2 -19173.358} C_VEL
LIN {X 0,Y 239.925,Z 468.661,A -85,B 0,C 180,E1 -19175.126,E2 -19175.126} C_VEL
LIN {X 0,Y 240.046,Z 467.827,A -85,B 0,C 180,E1 -19176.725,E2 -19176.725} C_VEL
LIN {X 0,Y 240.358,Z 466.514,A -85,B 0,C 180,E1 -19178.406,E2 -19178.406} C_VEL
LIN {X 0,Y 241.202,Z 463.551,A -85,B 0,C 180,E1 -19180.917,E2 -19180.917} C_VEL
LIN {X 0,Y 242.026,Z 460.878,A -85,B 0,C 180,E1 -19182.579,E2 -19182.579} C_VEL
LIN {X 0,Y 243.601,Z 455.682,A -85,B 0,C 180,E1 -19185.049,E2 -19185.049} C_VEL
LIN {X 0,Y 245.722,Z 448.893,A -85,B 0,C 180,E1 -19187.476,E2 -19187.476} C_VEL
LIN {X 0,Y 247.925,Z 441.497,A -85,B 0,C 180,E1 -19189.456,E2 -19189.456} C_VEL
LIN {X 0,Y 249.816,Z 434.234,A -85,B 0,C 180,E1 -19191.02,E2 -19191.02} C_VEL
LIN {X 0,Y 251.473,Z 427.707,A -85,B 0,C 180,E1 -19192.166,E2 -19192.166} C_VEL
LIN {X 0,Y 253.16,Z 419.837,A -85,B 0,C 180,E1 -19193.303,E2 -19193.303} C_VEL
LIN {X 0,Y 254.716,Z 411.75,A -85,B 0,C 180,E1 -19194.231,E2 -19194.231} C_VEL
LIN {X 0,Y 256.143,Z 403.134,A -85,B 0,C 180,E1 -19194.995,E2 -19194.995} C_VEL
LIN {X 0,Y 257.33,Z 393.916,A -85,B 0,C 180,E1 -19195.598,E2 -19195.598} C_VEL
LIN {X 0,Y 258.11,Z 384.471,A -85,B 0,C 180,E1 -19196.023,E2 -19196.023} C_VEL
LIN {X 0,Y 259.09,Z 357.343,A -85,B 0,C 180,E1 -19196.817,E2 -19196.817} C_VEL
LIN {X 0,Y 256.624,Z 340.416,A -85,B 0,C 180,E1 -19197.73,E2 -19197.73} C_VEL
LIN {X 0,Y 253.083,Z 322.491,A -85,B 0,C 180,E1 -19198.873,E2 -19198.873} C_VEL
LIN {X 0,Y 247.58,Z 310.545,A -85,B 0,C 180,E1 -19200.176,E2 -19200.176} C_VEL
LIN {X 0,Y 245.935,Z 306.775,A -85,B 0,C 180,E1 -19200.618,E2 -19200.618} C_VEL
LIN {X 0,Y 244.007,Z 298.078,A -85,B 0,C 180,E1 -19204.702,E2 -19204.702} C_VEL
LIN {X 0,Y 242.613,Z 292.586,A -85,B 0,C 180,E1 -19207.468,E2 -19207.468} C_VEL
LIN {X 0,Y 241.972,Z 290.154,A -85,B 0,C 180,E1 -19208.776,E2 -19208.776} C_VEL
LIN {X 0,Y 241.935,Z 290.159,A -85,B 0,C 180,E1 -19213.423,E2 -19213.423} C_VEL
LIN {X 0,Y 241.918,Z 290.158,A -85,B 0,C 180,E1 -19218.068,E2 -19218.068} C_VEL
LIN {X 0,Y 241.989,Z 290.154,A -85,B 0,C 180,E1 -19222.413,E2 -19222.413} C_VEL
LIN {X 0,Y 241.988,Z 290.153,A -85,B 0,C 180,E1 -19226.504,E2 -19226.504} C_VEL
LIN {X 0,Y 241.986,Z 290.153,A -85,B 0,C 180,E1 -19230.608,E2 -19230.608} C_VEL
LIN {X 0,Y 242.04,Z 290.138,A -85,B 0,C 180,E1 -19234.175,E2 -19234.175} C_VEL
LIN {X 0,Y 242.029,Z 290.136,A -85,B 0,C 180,E1 -19238.311,E2 -19238.311} C_VEL
LIN {X 0,Y 242.133,Z 290.123,A -85,B 0,C 180,E1 -19243.302,E2 -19243.302} C_VEL
LIN {X 0,Y 242.183,Z 290.114,A -85,B 0,C 180,E1 -19248.275,E2 -19248.275} C_VEL
LIN {X 0,Y 242.404,Z 290.097,A -85,B 0,C 180,E1 -19251.66,E2 -19251.66} C_VEL
LIN {X 0,Y 242.425,Z 290.087,A -85,B 0,C 180,E1 -19253.336,E2 -19253.336} C_VEL
LIN {X 0,Y 242.632,Z 290.064,A -85,B 0,C 180,E1 -19258.335,E2 -19258.335} C_VEL
LIN {X 0,Y 242.633,Z 290.065,A -85,B 0,C 180,E1 -19261.654,E2 -19261.654} C_VEL
LIN {X 0,Y 242.404,Z 290.093,A -85,B 0,C 180,E1 -19266.654,E2 -19266.654} C_VEL
LIN {X 0,Y 242.263,Z 290.108,A -85,B 0,C 180,E1 -19270.018,E2 -19270.018} C_VEL
LIN {X 0,Y 242.16,Z 290.123,A -85,B 0,C 180,E1 -19275.135,E2 -19275.135} C_VEL
LIN {X 0,Y 242.065,Z 290.143,A -85,B 0,C 180,E1 -19278.618,E2 -19278.618} C_VEL
LIN {X 0,Y 242.003,Z 290.151,A -85,B 0,C 180,E1 -19282.174,E2 -19282.174} C_VEL
LIN {X 0,Y 242.055,Z 290.143,A -85,B 0,C 180,E1 -19285.832,E2 -19285.832} C_VEL
LIN {X 0,Y 241.994,Z 290.153,A -85,B 0,C 180,E1 -19289.578,E2 -19289.578} C_VEL
LIN {X 0,Y 241.966,Z 290.158,A -85,B 0,C 180,E1 -19293.487,E2 -19293.487} C_VEL
LIN {X 0,Y 241.989,Z 290.148,A -85,B 0,C 180,E1 -19297.574,E2 -19297.574} C_VEL
LIN {X 0,Y 242.005,Z 290.148,A -85,B 0,C 180,E1 -19301.764,E2 -19301.764} C_VEL
LIN {X 0,Y 243.018,Z 293.016,A -85,B 0,C 180,E1 -19302.068,E2 -19302.068} C_VEL
LIN {X 0,Y 244.646,Z 295.216,A -85,B 0,C 180,E1 -19302.44,E2 -19302.44} C_VEL
LIN {X 0,Y 252.319,Z 308.399,A -85,B 0,C 180,E1 -19304.194,E2 -19304.194} C_VEL
LIN {X 0,Y 258.347,Z 321.385,A -85,B 0,C 180,E1 -19305.56,E2 -19305.56} C_VEL
LIN {X 0,Y 260.297,Z 326.197,A -85,B 0,C 180,E1 -19306.004,E2 -19306.004} C_VEL
LIN {X 0,Y 258.75,Z 364.976,A -85,B 0,C 180,E1 -19307.113,E2 -19307.113} C_VEL
LIN {X 0,Y 258.097,Z 374.179,A -85,B 0,C 180,E1 -19307.562,E2 -19307.562} C_VEL
LIN {X 0,Y 257.142,Z 383.5,A -85,B 0,C 180,E1 -19308.226,E2 -19308.226} C_VEL
LIN {X 0,Y 255.651,Z 394.003,A -85,B 0,C 180,E1 -19309.24,E2 -19309.24} C_VEL
LIN {X 0,Y 253.677,Z 404.516,A -85,B 0,C 180,E1 -19310.646,E2 -19310.646} C_VEL
LIN {X 0,Y 252.133,Z 411.451,A -85,B 0,C 180,E1 -19311.808,E2 -19311.808} C_VEL
LIN {X 0,Y 250.211,Z 418.938,A -85,B 0,C 180,E1 -19313.354,E2 -19313.354} C_VEL
LIN {X 0,Y 248.429,Z 425.298,A -85,B 0,C 180,E1 -19314.981,E2 -19314.981} C_VEL
LIN {X 0,Y 246.698,Z 430.888,A -85,B 0,C 180,E1 -19316.743,E2 -19316.743} C_VEL
LIN {X 0,Y 245.227,Z 435.306,A -85,B 0,C 180,E1 -19318.465,E2 -19318.465} C_VEL
LIN {X 0,Y 243.69,Z 439.697,A -85,B 0,C 180,E1 -19320.641,E2 -19320.641} C_VEL
LIN {X 0,Y 242.196,Z 443.561,A -85,B 0,C 180,E1 -19323.271,E2 -19323.271} C_VEL
LIN {X 0,Y 241.081,Z 445.912,A -85,B 0,C 180,E1 -19325.913,E2 -19325.913} C_VEL
LIN {X 0,Y 240.547,Z 446.835,A -85,B 0,C 180,E1 -19327.678,E2 -19327.678} C_VEL
LIN {X 0,Y 240.16,Z 447.144,A -85,B 0,C 180,E1 -19329.442,E2 -19329.442} C_VEL
LIN {X 0,Y 239.89,Z 446.888,A -85,B 0,C 180,E1 -19331.2,E2 -19331.2} C_VEL
LIN {X 0,Y 239.76,Z 446.121,A -85,B 0,C 180,E1 -19332.955,E2 -19332.955} C_VEL
LIN {X 0,Y 239.829,Z 444.332,A -85,B 0,C 180,E1 -19335.219,E2 -19335.219} C_VEL
LIN {X 0,Y 240.068,Z 441.804,A -85,B 0,C 180,E1 -19337.317,E2 -19337.317} C_VEL
LIN {X 0,Y 240.362,Z 439.04,A -85,B 0,C 180,E1 -19339.044,E2 -19339.044} C_VEL
LIN {X 0,Y 240.744,Z 435.629,A -85,B 0,C 180,E1 -19340.761,E2 -19340.761} C_VEL
LIN {X 0,Y 241.369,Z 430.709,A -85,B 0,C 180,E1 -19342.741,E2 -19342.741} C_VEL
LIN {X 0,Y 241.951,Z 425.052,A -85,B 0,C 180,E1 -19344.583,E2 -19344.583} C_VEL
LIN {X 0,Y 242.765,Z 418.716,A -85,B 0,C 180,E1 -19346.266,E2 -19346.266} C_VEL
LIN {X 0,Y 243.559,Z 412.053,A -85,B 0,C 180,E1 -19347.726,E2 -19347.726} C_VEL
LIN {X 0,Y 244.528,Z 403.96,A -85,B 0,C 180,E1 -19349.177,E2 -19349.177} C_VEL
LIN {X 0,Y 245.619,Z 393.319,A -85,B 0,C 180,E1 -19350.677,E2 -19350.677} C_VEL
LIN {X 0,Y 246.367,Z 383.047,A -85,B 0,C 180,E1 -19351.732,E2 -19351.732} C_VEL
LIN {X 0,Y 246.952,Z 373.384,A -85,B 0,C 180,E1 -19352.456,E2 -19352.456} C_VEL
LIN {X 0,Y 247.307,Z 363.974,A -85,B 0,C 180,E1 -19352.938,E2 -19352.938} C_VEL
LIN {X 0,Y 248.493,Z 313.52,A -85,B 0,C 180,E1 -19354.426,E2 -19354.426} C_VEL
LIN {X 0,Y 246.7,Z 303.05,A -85,B 0,C 180,E1 -19354.865,E2 -19354.865} C_VEL
LIN {X 0,Y 242.286,Z 290.118,A -85,B 0,C 180,E1 -19355.58,E2 -19355.58} C_VEL
LIN {X 0,Y 242.369,Z 290.104,A -85,B 0,C 180,E1 -19358.337,E2 -19358.337} C_VEL
LIN {X 0,Y 242.111,Z 290.14,A -85,B 0,C 180,E1 -19363.428,E2 -19363.428} C_VEL
LIN {X 0,Y 242.114,Z 290.137,A -85,B 0,C 180,E1 -19366.875,E2 -19366.875} C_VEL
LIN {X 0,Y 241.998,Z 290.154,A -85,B 0,C 180,E1 -19371.689,E2 -19371.689} C_VEL
LIN {X 0,Y 242.006,Z 290.152,A -85,B 0,C 180,E1 -19375.824,E2 -19375.824} C_VEL
LIN {X 0,Y 241.942,Z 290.158,A -85,B 0,C 180,E1 -19379.593,E2 -19379.593} C_VEL
LIN {X 0,Y 241.954,Z 290.155,A -85,B 0,C 180,E1 -19383.497,E2 -19383.497} C_VEL
LIN {X 0,Y 241.96,Z 290.157,A -85,B 0,C 180,E1 -19387.588,E2 -19387.588} C_VEL
LIN {X 0,Y 241.901,Z 290.164,A -85,B 0,C 180,E1 -19391.931,E2 -19391.931} C_VEL
LIN {X 0,Y 241.906,Z 290.162,A -85,B 0,C 180,E1 -19396.579,E2 -19396.579} C_VEL
LIN {X 0,Y 241.94,Z 290.156,A -85,B 0,C 180,E1 -19400.286,E2 -19400.286} C_VEL
LIN {X 0,Y 241.974,Z 290.154,A -85,B 0,C 180,E1 -19404.495,E2 -19404.495} C_VEL
LIN {X 0,Y 241.94,Z 290.157,A -85,B 0,C 180,E1 -19408.482,E2 -19408.482} C_VEL
LIN {X 0,Y 241.957,Z 290.157,A -85,B 0,C 180,E1 -19412.314,E2 -19412.314} C_VEL
LIN {X 0,Y 242.017,Z 290.145,A -85,B 0,C 180,E1 -19416.019,E2 -19416.019} C_VEL
LIN {X 0,Y 242.201,Z 290.107,A -85,B 0,C 180,E1 -19421.392,E2 -19421.392} C_VEL
LIN {X 0,Y 242.309,Z 290.091,A -85,B 0,C 180,E1 -19422.123,E2 -19422.123} C_VEL
LIN {X 0,Y 244.403,Z 311.012,A -85,B 0,C 180,E1 -19423.16,E2 -19423.16} C_VEL
LIN {X 0,Y 242.992,Z 366.657,A -85,B 0,C 180,E1 -19425.935,E2 -19425.935} C_VEL
LIN {X 0,Y 242.612,Z 377.109,A -85,B 0,C 180,E1 -19426.713,E2 -19426.713} C_VEL
LIN {X 0,Y 242.226,Z 388.569,A -85,B 0,C 180,E1 -19427.863,E2 -19427.863} C_VEL
LIN {X 0,Y 241.651,Z 399.36,A -85,B 0,C 180,E1 -19429.321,E2 -19429.321} C_VEL
LIN {X 0,Y 241.144,Z 409.286,A -85,B 0,C 180,E1 -19430.993,E2 -19430.993} C_VEL
LIN {X 0,Y 240.741,Z 418.27,A -85,B 0,C 180,E1 -19432.921,E2 -19432.921} C_VEL
LIN {X 0,Y 240.368,Z 425.983,A -85,B 0,C 180,E1 -19434.973,E2 -19434.973} C_VEL
LIN {X 0,Y 240.168,Z 432.379,A -85,B 0,C 180,E1 -19437.07,E2 -19437.07} C_VEL
LIN {X 0,Y 239.965,Z 437.633,A -85,B 0,C 180,E1 -19439.28,E2 -19439.28} C_VEL
LIN {X 0,Y 240.097,Z 441.962,A -85,B 0,C 180,E1 -19441.683,E2 -19441.683} C_VEL
LIN {X 0,Y 240.381,Z 444.329,A -85,B 0,C 180,E1 -19443.357,E2 -19443.357} C_VEL
LIN {X 0,Y 240.81,Z 446.136,A -85,B 0,C 180,E1 -19445.028,E2 -19445.028} C_VEL
LIN {X 0,Y 241.171,Z 446.982,A -85,B 0,C 180,E1 -19446.195,E2 -19446.195} C_VEL
LIN {X 0,Y 240.815,Z 447.622,A -85,B 0,C 180,E1 -19447.129,E2 -19447.129} C_VEL
LIN {X 0,Y 238.528,Z 448.336,A -85,B 0,C 180,E1 -19448.644,E2 -19448.644} C_VEL
LIN {X 0,Y 236.482,Z 448.712,A -85,B 0,C 180,E1 -19450.193,E2 -19450.193} C_VEL
LIN {X 0,Y 236.503,Z 448.699,A -85,B 0,C 180,E1 -19451.154,E2 -19451.154} C_VEL
LIN {X 0,Y 238.525,Z 448.037,A -85,B 0,C 180,E1 -19453.639,E2 -19453.639} C_VEL
LIN {X 0,Y 240.294,Z 446.945,A -85,B 0,C 180,E1 -19455.267,E2 -19455.267} C_VEL
LIN {X 0,Y 243.173,Z 444.327,A -85,B 0,C 180,E1 -19457.671,E2 -19457.671} C_VEL
LIN {X 0,Y 246.587,Z 440.461,A -85,B 0,C 180,E1 -19460.004,E2 -19460.004} C_VEL
LIN {X 0,Y 250.419,Z 435.171,A -85,B 0,C 180,E1 -19462.269,E2 -19462.269} C_VEL
LIN {X 0,Y 253.924,Z 429.472,A -85,B 0,C 180,E1 -19464.099,E2 -19464.099} C_VEL
LIN {X 0,Y 257.716,Z 422.5,A -85,B 0,C 180,E1 -19465.874,E2 -19465.874} C_VEL
LIN {X 0,Y 261.835,Z 413.884,A -85,B 0,C 180,E1 -19467.586,E2 -19467.586} C_VEL
LIN {X 0,Y 265.694,Z 404.001,A -85,B 0,C 180,E1 -19469.085,E2 -19469.085} C_VEL
LIN {X 0,Y 269.374,Z 393.161,A -85,B 0,C 180,E1 -19470.369,E2 -19470.369} C_VEL
LIN {X 0,Y 272.202,Z 382.516,A -85,B 0,C 180,E1 -19471.31,E2 -19471.31} C_VEL
LIN {X 0,Y 274.527,Z 371.647,A -85,B 0,C 180,E1 -19472.028,E2 -19472.028} C_VEL
LIN {X 0,Y 278.139,Z 350.154,A -85,B 0,C 180,E1 -19473.101,E2 -19473.101} C_VEL
LIN {X 0,Y 275.689,Z 344.475,A -85,B 0,C 180,E1 -19475.085,E2 -19475.085} C_VEL
LIN {X 0,Y 273.809,Z 340.763,A -85,B 0,C 180,E1 -19476.866,E2 -19476.866} C_VEL
LIN {X 0,Y 272.317,Z 338.021,A -85,B 0,C 180,E1 -19478.624,E2 -19478.624} C_VEL
LIN {X 0,Y 270.841,Z 335.471,A -85,B 0,C 180,E1 -19481.191,E2 -19481.191} C_VEL
LIN {X 0,Y 270.171,Z 334.693,A -85,B 0,C 180,E1 -19483.25,E2 -19483.25} C_VEL
LIN {X 0,Y 270.181,Z 334.887,A -85,B 0,C 180,E1 -19486.127,E2 -19486.127} C_VEL
LIN {X 0,Y 270.884,Z 335.829,A -85,B 0,C 180,E1 -19488.215,E2 -19488.215} C_VEL
LIN {X 0,Y 272.938,Z 340.088,A -85,B 0,C 180,E1 -19491.577,E2 -19491.577} C_VEL
LIN {X 0,Y 274.61,Z 343.427,A -85,B 0,C 180,E1 -19493.365,E2 -19493.365} C_VEL
LIN {X 0,Y 276.827,Z 348.069,A -85,B 0,C 180,E1 -19495.274,E2 -19495.274} C_VEL
LIN {X 0,Y 276.331,Z 359.865,A -85,B 0,C 180,E1 -19496.545,E2 -19496.545} C_VEL
LIN {X 0,Y 275.899,Z 365.456,A -85,B 0,C 180,E1 -19497.045,E2 -19497.045} C_VEL
LIN {X 0,Y 271.94,Z 388.237,A -85,B 0,C 180,E1 -19498.226,E2 -19498.226} C_VEL
LIN {X 0,Y 269.151,Z 398.966,A -85,B 0,C 180,E1 -19498.955,E2 -19498.955} C_VEL
LIN {X 0,Y 265.888,Z 409.189,A -85,B 0,C 180,E1 -19499.853,E2 -19499.853} C_VEL
LIN {X 0,Y 261.782,Z 420.008,A -85,B 0,C 180,E1 -19501.102,E2 -19501.102} C_VEL
LIN {X 0,Y 258.004,Z 428.676,A -85,B 0,C 180,E1 -19502.414,E2 -19502.414} C_VEL
LIN {X 0,Y 254.493,Z 435.876,A -85,B 0,C 180,E1 -19503.778,E2 -19503.778} C_VEL
LIN {X 0,Y 250.479,Z 443.361,A -85,B 0,C 180,E1 -19505.552,E2 -19505.552} C_VEL
LIN {X 0,Y 246.211,Z 450.473,A -85,B 0,C 180,E1 -19507.776,E2 -19507.776} C_VEL
LIN {X 0,Y 243.117,Z 455.133,A -85,B 0,C 180,E1 -19509.702,E2 -19509.702} C_VEL
LIN {X 0,Y 239.906,Z 459.491,A -85,B 0,C 180,E1 -19512.085,E2 -19512.085} C_VEL
LIN {X 0,Y 238.896,Z 460.74,A -85,B 0,C 180,E1 -19512.891,E2 -19512.891} C_VEL
LIN {X 0,Y 237.33,Z 462.616,A -85,B 0,C 180,E1 -19514.543,E2 -19514.543} C_VEL
LIN {X 0,Y 235.947,Z 464.011,A -85,B 0,C 180,E1 -19516.214,E2 -19516.214} C_VEL
LIN {X 0,Y 234.856,Z 464.966,A -85,B 0,C 180,E1 -19517.908,E2 -19517.908} C_VEL
LIN {X 0,Y 234.007,Z 465.463,A -85,B 0,C 180,E1 -19519.618,E2 -19519.618} C_VEL
LIN {X 0,Y 233.41,Z 465.378,A -85,B 0,C 180,E1 -19521.341,E2 -19521.341} C_VEL
LIN {X 0,Y 233.069,Z 464.169,A -85,B 0,C 180,E1 -19524.353,E2 -19524.353} C_VEL
LIN {X 0,Y 233.102,Z 463.347,A -85,B 0,C 180,E1 -19525.546,E2 -19525.546} C_VEL
LIN {X 0,Y 232.954,Z 466.432,A -85,B 0,C 180,E1 -19528.271,E2 -19528.271} C_VEL
LIN {X 0,Y 232.953,Z 467.684,A -85,B 0,C 180,E1 -19530,E2 -19530} C_VEL
LIN {X 0,Y 232.909,Z 468.451,A -85,B 0,C 180,E1 -19531.729,E2 -19531.729} C_VEL
LIN {X 0,Y 232.827,Z 468.71,A -85,B 0,C 180,E1 -19533.461,E2 -19533.461} C_VEL
LIN {X 0,Y 232.854,Z 468.383,A -85,B 0,C 180,E1 -19535.195,E2 -19535.195} C_VEL
LIN {X 0,Y 232.992,Z 467.592,A -85,B 0,C 180,E1 -19536.93,E2 -19536.93} C_VEL
LIN {X 0,Y 233.317,Z 466.343,A -85,B 0,C 180,E1 -19538.662,E2 -19538.662} C_VEL
LIN {X 0,Y 234.209,Z 463.445,A -85,B 0,C 180,E1 -19541.247,E2 -19541.247} C_VEL
LIN {X 0,Y 235.593,Z 459.311,A -85,B 0,C 180,E1 -19543.806,E2 -19543.806} C_VEL
LIN {X 0,Y 237.454,Z 453.76,A -85,B 0,C 180,E1 -19546.33,E2 -19546.33} C_VEL
LIN {X 0,Y 239.41,Z 447.711,A -85,B 0,C 180,E1 -19548.395,E2 -19548.395} C_VEL
LIN {X 0,Y 241.272,Z 441.829,A -85,B 0,C 180,E1 -19550.015,E2 -19550.015} C_VEL
LIN {X 0,Y 243.23,Z 434.705,A -85,B 0,C 180,E1 -19551.617,E2 -19551.617} C_VEL
LIN {X 0,Y 245.241,Z 427.122,A -85,B 0,C 180,E1 -19552.983,E2 -19552.983} C_VEL
LIN {X 0,Y 246.997,Z 419.207,A -85,B 0,C 180,E1 -19554.143,E2 -19554.143} C_VEL
LIN {X 0,Y 248.65,Z 411.05,A -85,B 0,C 180,E1 -19555.085,E2 -19555.085} C_VEL
LIN {X 0,Y 250.089,Z 402.747,A -85,B 0,C 180,E1 -19555.828,E2 -19555.828} C_VEL
LIN {X 0,Y 251.334,Z 393.144,A -85,B 0,C 180,E1 -19556.466,E2 -19556.466} C_VEL
LIN {X 0,Y 252.169,Z 383.652,A -85,B 0,C 180,E1 -19556.887,E2 -19556.887} C_VEL
LIN {X 0,Y 253.081,Z 358.108,A -85,B 0,C 180,E1 -19557.655,E2 -19557.655} C_VEL
LIN {X 0,Y 250.248,Z 338.899,A -85,B 0,C 180,E1 -19558.746,E2 -19558.746} C_VEL
LIN {X 0,Y 247.316,Z 324.89,A -85,B 0,C 180,E1 -19559.708,E2 -19559.708} C_VEL
LIN {X 0,Y 240.659,Z 310.608,A -85,B 0,C 180,E1 -19561.374,E2 -19561.374} C_VEL
LIN {X 0,Y 238.605,Z 306.295,A -85,B 0,C 180,E1 -19561.962,E2 -19561.962} C_VEL
LIN {X 0,Y 236.876,Z 298.357,A -85,B 0,C 180,E1 -19565.871,E2 -19565.871} C_VEL
LIN {X 0,Y 234.934,Z 291.033,A -85,B 0,C 180,E1 -19569.887,E2 -19569.887} C_VEL
LIN {X 0,Y 234.893,Z 291.032,A -85,B 0,C 180,E1 -19574.098,E2 -19574.098} C_VEL
LIN {X 0,Y 234.861,Z 291.042,A -85,B 0,C 180,E1 -19578.822,E2 -19578.822} C_VEL
LIN {X 0,Y 234.928,Z 291.025,A -85,B 0,C 180,E1 -19581.075,E2 -19581.075} C_VEL
LIN {X 0,Y 234.931,Z 291.024,A -85,B 0,C 180,E1 -19585.357,E2 -19585.357} C_VEL
LIN {X 0,Y 234.907,Z 291.026,A -85,B 0,C 180,E1 -19589.424,E2 -19589.424} C_VEL
LIN {X 0,Y 234.977,Z 291.017,A -85,B 0,C 180,E1 -19593.802,E2 -19593.802} C_VEL
LIN {X 0,Y 234.997,Z 291.011,A -85,B 0,C 180,E1 -19598.963,E2 -19598.963} C_VEL
LIN {X 0,Y 235.069,Z 291.003,A -85,B 0,C 180,E1 -19603.081,E2 -19603.081} C_VEL
LIN {X 0,Y 235.115,Z 290.997,A -85,B 0,C 180,E1 -19607.917,E2 -19607.917} C_VEL
LIN {X 0,Y 235.335,Z 290.977,A -85,B 0,C 180,E1 -19611.407,E2 -19611.407} C_VEL
LIN {X 0,Y 235.375,Z 290.967,A -85,B 0,C 180,E1 -19613.135,E2 -19613.135} C_VEL
LIN {X 0,Y 235.591,Z 290.941,A -85,B 0,C 180,E1 -19618.285,E2 -19618.285} C_VEL
LIN {X 0,Y 235.592,Z 290.943,A -85,B 0,C 180,E1 -19621.704,E2 -19621.704} C_VEL
LIN {X 0,Y 235.356,Z 290.973,A -85,B 0,C 180,E1 -19626.854,E2 -19626.854} C_VEL
LIN {X 0,Y 235.21,Z 290.985,A -85,B 0,C 180,E1 -19630.322,E2 -19630.322} C_VEL
LIN {X 0,Y 235.107,Z 290.999,A -85,B 0,C 180,E1 -19635.601,E2 -19635.601} C_VEL
LIN {X 0,Y 235.001,Z 291.021,A -85,B 0,C 180,E1 -19639.2,E2 -19639.2} C_VEL
LIN {X 0,Y 234.951,Z 291.03,A -85,B 0,C 180,E1 -19642.877,E2 -19642.877} C_VEL
LIN {X 0,Y 234.956,Z 291.032,A -85,B 0,C 180,E1 -19646.652,E2 -19646.652} C_VEL
LIN {X 0,Y 234.908,Z 291.036,A -85,B 0,C 180,E1 -19650.563,E2 -19650.563} C_VEL
LIN {X 0,Y 234.918,Z 291.022,A -85,B 0,C 180,E1 -19654.632,E2 -19654.632} C_VEL
LIN {X 0,Y 234.949,Z 291.028,A -85,B 0,C 180,E1 -19658.947,E2 -19658.947} C_VEL
LIN {X 0,Y 234.947,Z 291.019,A -85,B 0,C 180,E1 -19660.437,E2 -19660.437} C_VEL
LIN {X 0,Y 235.983,Z 293.938,A -85,B 0,C 180,E1 -19660.784,E2 -19660.784} C_VEL
LIN {X 0,Y 237.64,Z 296.142,A -85,B 0,C 180,E1 -19661.19,E2 -19661.19} C_VEL
LIN {X 0,Y 246.14,Z 310.242,A -85,B 0,C 180,E1 -19663.248,E2 -19663.248} C_VEL
LIN {X 0,Y 252.372,Z 323.429,A -85,B 0,C 180,E1 -19664.724,E2 -19664.724} C_VEL
LIN {X 0,Y 254.315,Z 328.003,A -85,B 0,C 180,E1 -19665.18,E2 -19665.18} C_VEL
LIN {X 0,Y 252.726,Z 365.959,A -85,B 0,C 180,E1 -19666.295,E2 -19666.295} C_VEL
LIN {X 0,Y 252.023,Z 375.173,A -85,B 0,C 180,E1 -19666.767,E2 -19666.767} C_VEL
LIN {X 0,Y 250.89,Z 385.319,A -85,B 0,C 180,E1 -19667.523,E2 -19667.523} C_VEL
LIN {X 0,Y 249.052,Z 396.698,A -85,B 0,C 180,E1 -19668.73,E2 -19668.73} C_VEL
LIN {X 0,Y 247.437,Z 404.869,A -85,B 0,C 180,E1 -19669.875,E2 -19669.875} C_VEL
LIN {X 0,Y 245.577,Z 412.725,A -85,B 0,C 180,E1 -19671.243,E2 -19671.243} C_VEL
LIN {X 0,Y 243.697,Z 419.641,A -85,B 0,C 180,E1 -19672.727,E2 -19672.727} C_VEL
LIN {X 0,Y 241.739,Z 426.233,A -85,B 0,C 180,E1 -19674.48,E2 -19674.48} C_VEL
LIN {X 0,Y 239.618,Z 432.695,A -85,B 0,C 180,E1 -19676.638,E2 -19676.638} C_VEL
LIN {X 0,Y 237.697,Z 438.091,A -85,B 0,C 180,E1 -19679.017,E2 -19679.017} C_VEL
LIN {X 0,Y 236.018,Z 442.234,A -85,B 0,C 180,E1 -19681.547,E2 -19681.547} C_VEL
LIN {X 0,Y 234.804,Z 444.911,A -85,B 0,C 180,E1 -19683.872,E2 -19683.872} C_VEL
LIN {X 0,Y 234.261,Z 446.041,A -85,B 0,C 180,E1 -19685.165,E2 -19685.165} C_VEL
LIN {X 0,Y 233.631,Z 447.021,A -85,B 0,C 180,E1 -19686.98,E2 -19686.98} C_VEL
LIN {X 0,Y 233.135,Z 447.469,A -85,B 0,C 180,E1 -19689.129,E2 -19689.129} C_VEL
LIN {X 0,Y 232.706,Z 446.659,A -85,B 0,C 180,E1 -19692.422,E2 -19692.422} C_VEL
LIN {X 0,Y 232.744,Z 444.725,A -85,B 0,C 180,E1 -19695.049,E2 -19695.049} C_VEL
LIN {X 0,Y 232.917,Z 442.615,A -85,B 0,C 180,E1 -19696.921,E2 -19696.921} C_VEL
LIN {X 0,Y 233.391,Z 438.423,A -85,B 0,C 180,E1 -19699.591,E2 -19699.591} C_VEL
LIN {X 0,Y 234.066,Z 432.88,A -85,B 0,C 180,E1 -19702.186,E2 -19702.186} C_VEL
LIN {X 0,Y 234.753,Z 426.538,A -85,B 0,C 180,E1 -19704.417,E2 -19704.417} C_VEL
LIN {X 0,Y 235.603,Z 420.422,A -85,B 0,C 180,E1 -19706.152,E2 -19706.152} C_VEL
LIN {X 0,Y 236.508,Z 412.995,A -85,B 0,C 180,E1 -19707.872,E2 -19707.872} C_VEL
LIN {X 0,Y 237.449,Z 405.041,A -85,B 0,C 180,E1 -19709.364,E2 -19709.364} C_VEL
LIN {X 0,Y 238.429,Z 396.164,A -85,B 0,C 180,E1 -19710.697,E2 -19710.697} C_VEL
LIN {X 0,Y 239.406,Z 385.037,A -85,B 0,C 180,E1 -19711.972,E2 -19711.972} C_VEL
LIN {X 0,Y 240.045,Z 374.053,A -85,B 0,C 180,E1 -19712.842,E2 -19712.842} C_VEL
LIN {X 0,Y 240.442,Z 364.424,A -85,B 0,C 180,E1 -19713.352,E2 -19713.352} C_VEL
LIN {X 0,Y 241.577,Z 313.553,A -85,B 0,C 180,E1 -19714.902,E2 -19714.902} C_VEL
LIN {X 0,Y 240.104,Z 305.081,A -85,B 0,C 180,E1 -19715.271,E2 -19715.271} C_VEL
LIN {X 0,Y 235.279,Z 290.99,A -85,B 0,C 180,E1 -19716.108,E2 -19716.108} C_VEL
LIN {X 0,Y 235.258,Z 290.994,A -85,B 0,C 180,E1 -19719.703,E2 -19719.703} C_VEL
LIN {X 0,Y 235.066,Z 291.016,A -85,B 0,C 180,E1 -19725.61,E2 -19725.61} C_VEL
LIN {X 0,Y 234.976,Z 291.029,A -85,B 0,C 180,E1 -19729.209,E2 -19729.209} C_VEL
LIN {X 0,Y 234.92,Z 291.034,A -85,B 0,C 180,E1 -19732.887,E2 -19732.887} C_VEL
LIN {X 0,Y 234.918,Z 291.033,A -85,B 0,C 180,E1 -19736.664,E2 -19736.664} C_VEL
LIN {X 0,Y 234.872,Z 291.035,A -85,B 0,C 180,E1 -19740.577,E2 -19740.577} C_VEL
LIN {X 0,Y 234.899,Z 291.034,A -85,B 0,C 180,E1 -19744.644,E2 -19744.644} C_VEL
LIN {X 0,Y 234.89,Z 291.034,A -85,B 0,C 180,E1 -19748.94,E2 -19748.94} C_VEL
LIN {X 0,Y 234.851,Z 291.043,A -85,B 0,C 180,E1 -19753.495,E2 -19753.495} C_VEL
LIN {X 0,Y 234.859,Z 291.04,A -85,B 0,C 180,E1 -19756.517,E2 -19756.517} C_VEL
LIN {X 0,Y 234.902,Z 291.032,A -85,B 0,C 180,E1 -19761.084,E2 -19761.084} C_VEL
LIN {X 0,Y 234.916,Z 291.034,A -85,B 0,C 180,E1 -19765.368,E2 -19765.368} C_VEL
LIN {X 0,Y 234.886,Z 291.036,A -85,B 0,C 180,E1 -19769.433,E2 -19769.433} C_VEL
LIN {X 0,Y 234.959,Z 291.03,A -85,B 0,C 180,E1 -19773.813,E2 -19773.813} C_VEL
LIN {X 0,Y 235.004,Z 291.006,A -85,B 0,C 180,E1 -19778.976,E2 -19778.976} C_VEL
LIN {X 0,Y 235.255,Z 290.969,A -85,B 0,C 180,E1 -19782.097,E2 -19782.097} C_VEL
LIN {X 0,Y 237.322,Z 310.57,A -85,B 0,C 180,E1 -19783.113,E2 -19783.113} C_VEL
LIN {X 0,Y 235.914,Z 366.671,A -85,B 0,C 180,E1 -19786.054,E2 -19786.054} C_VEL
LIN {X 0,Y 235.545,Z 377.109,A -85,B 0,C 180,E1 -19786.856,E2 -19786.856} C_VEL
LIN {X 0,Y 235.176,Z 387.703,A -85,B 0,C 180,E1 -19787.931,E2 -19787.931} C_VEL
LIN {X 0,Y 234.615,Z 398.794,A -85,B 0,C 180,E1 -19789.434,E2 -19789.434} C_VEL
LIN {X 0,Y 234.168,Z 407.692,A -85,B 0,C 180,E1 -19790.94,E2 -19790.94} C_VEL
LIN {X 0,Y 233.717,Z 417.112,A -85,B 0,C 180,E1 -19792.903,E2 -19792.903} C_VEL
LIN {X 0,Y 233.326,Z 424.385,A -85,B 0,C 180,E1 -19794.821,E2 -19794.821} C_VEL
LIN {X 0,Y 233.251,Z 429.846,A -85,B 0,C 180,E1 -19796.551,E2 -19796.551} C_VEL
LIN {X 0,Y 232.993,Z 434.395,A -85,B 0,C 180,E1 -19798.277,E2 -19798.277} C_VEL
LIN {X 0,Y 232.949,Z 439.842,A -85,B 0,C 180,E1 -19800.87,E2 -19800.87} C_VEL
LIN {X 0,Y 233.325,Z 443.956,A -85,B 0,C 180,E1 -19803.459,E2 -19803.459} C_VEL
LIN {X 0,Y 233.749,Z 445.887,A -85,B 0,C 180,E1 -19805.18,E2 -19805.18} C_VEL
LIN {X 0,Y 234.299,Z 447.309,A -85,B 0,C 180,E1 -19806.896,E2 -19806.896} C_VEL
LIN {X 0,Y 234.946,Z 448.271,A -85,B 0,C 180,E1 -19808.607,E2 -19808.607} C_VEL
LIN {X 0,Y 235.819,Z 448.759,A -85,B 0,C 180,E1 -19810.306,E2 -19810.306} C_VEL
LIN {X 0,Y 236.503,Z 448.699,A -85,B 0,C 180,E1 -19811.154,E2 -19811.154} C_VEL
LIN {X 0,Y 236.634,Z 448.68,A -85,B 0,C 180,E1 -19812.119,E2 -19812.119} C_VEL
LIN {X 0,Y 235.153,Z 448.586,A -85,B 0,C 180,E1 -19813.722,E2 -19813.722} C_VEL
LIN {X 0,Y 233.823,Z 448.15,A -85,B 0,C 180,E1 -19815.336,E2 -19815.336} C_VEL
LIN {X 0,Y 234.184,Z 447.524,A -85,B 0,C 180,E1 -19816.295,E2 -19816.295} C_VEL
LIN {X 0,Y 237.66,Z 444.691,A -85,B 0,C 180,E1 -19818.988,E2 -19818.988} C_VEL
LIN {X 0,Y 241.424,Z 440.823,A -85,B 0,C 180,E1 -19821.344,E2 -19821.344} C_VEL
LIN {X 0,Y 245.566,Z 435.472,A -85,B 0,C 180,E1 -19823.625,E2 -19823.625} C_VEL
LIN {X 0,Y 249.352,Z 429.824,A -85,B 0,C 180,E1 -19825.461,E2 -19825.461} C_VEL
LIN {X 0,Y 253.411,Z 422.839,A -85,B 0,C 180,E1 -19827.237,E2 -19827.237} C_VEL
LIN {X 0,Y 258.246,Z 413.227,A -85,B 0,C 180,E1 -19829.112,E2 -19829.112} C_VEL
LIN {X 0,Y 261.936,Z 404.476,A -85,B 0,C 180,E1 -19830.431,E2 -19830.431} C_VEL
LIN {X 0,Y 265.813,Z 393.578,A -85,B 0,C 180,E1 -19831.705,E2 -19831.705} C_VEL
LIN {X 0,Y 268.751,Z 383.368,A -85,B 0,C 180,E1 -19832.611,E2 -19832.611} C_VEL
LIN {X 0,Y 271.108,Z 373.193,A -85,B 0,C 180,E1 -19833.301,E2 -19833.301} C_VEL
LIN {X 0,Y 274.587,Z 354.307,A -85,B 0,C 180,E1 -19834.228,E2 -19834.228} C_VEL
LIN {X 0,Y 272.79,Z 350.06,A -85,B 0,C 180,E1 -19835.886,E2 -19835.886} C_VEL
LIN {X 0,Y 271.514,Z 347.198,A -85,B 0,C 180,E1 -19837.271,E2 -19837.271} C_VEL
LIN {X 0,Y 270.269,Z 344.721,A -85,B 0,C 180,E1 -19838.861,E2 -19838.861} C_VEL
LIN {X 0,Y 268.873,Z 342.166,A -85,B 0,C 180,E1 -19841.554,E2 -19841.554} C_VEL
LIN {X 0,Y 268.399,Z 341.639,A -85,B 0,C 180,E1 -19842.911,E2 -19842.911} C_VEL
LIN {X 0,Y 268.329,Z 341.698,A -85,B 0,C 180,E1 -19845.935,E2 -19845.935} C_VEL
LIN {X 0,Y 268.925,Z 342.494,A -85,B 0,C 180,E1 -19847.916,E2 -19847.916} C_VEL
LIN {X 0,Y 270.871,Z 346.931,A -85,B 0,C 180,E1 -19851.416,E2 -19851.416} C_VEL
LIN {X 0,Y 272.27,Z 350.005,A -85,B 0,C 180,E1 -19853.025,E2 -19853.025} C_VEL
LIN {X 0,Y 273.662,Z 353.008,A -85,B 0,C 180,E1 -19854.322,E2 -19854.322} C_VEL
LIN {X 0,Y 272.727,Z 365.748,A -85,B 0,C 180,E1 -19855.681,E2 -19855.681} C_VEL
LIN {X 0,Y 269.114,Z 385.762,A -85,B 0,C 180,E1 -19856.741,E2 -19856.741} C_VEL
LIN {X 0,Y 265.757,Z 398.335,A -85,B 0,C 180,E1 -19857.576,E2 -19857.576} C_VEL
LIN {X 0,Y 261.673,Z 410.395,A -85,B 0,C 180,E1 -19858.642,E2 -19858.642} C_VEL
LIN {X 0,Y 257.376,Z 420.744,A -85,B 0,C 180,E1 -19859.883,E2 -19859.883} C_VEL
LIN {X 0,Y 253.84,Z 428.194,A -85,B 0,C 180,E1 -19861.019,E2 -19861.019} C_VEL
LIN {X 0,Y 249.236,Z 437.004,A -85,B 0,C 180,E1 -19862.727,E2 -19862.727} C_VEL
LIN {X 0,Y 245.016,Z 444.156,A -85,B 0,C 180,E1 -19864.516,E2 -19864.516} C_VEL
LIN {X 0,Y 241.906,Z 448.886,A -85,B 0,C 180,E1 -19866,E2 -19866} C_VEL
LIN {X 0,Y 237.787,Z 454.579,A -85,B 0,C 180,E1 -19868.318,E2 -19868.318} C_VEL
LIN {X 0,Y 234.278,Z 458.923,A -85,B 0,C 180,E1 -19870.732,E2 -19870.732} C_VEL
LIN {X 0,Y 232.132,Z 461.145,A -85,B 0,C 180,E1 -19872.376,E2 -19872.376} C_VEL
LIN {X 0,Y 230.493,Z 462.892,A -85,B 0,C 180,E1 -19874.072,E2 -19874.072} C_VEL
LIN {X 0,Y 229.072,Z 464.085,A -85,B 0,C 180,E1 -19875.792,E2 -19875.792} C_VEL
LIN {X 0,Y 227.927,Z 464.745,A -85,B 0,C 180,E1 -19877.535,E2 -19877.535} C_VEL
LIN {X 0,Y 227.04,Z 464.983,A -85,B 0,C 180,E1 -19879.296,E2 -19879.296} C_VEL
LIN {X 0,Y 226.417,Z 464.784,A -85,B 0,C 180,E1 -19881.071,E2 -19881.071} C_VEL
LIN {X 0,Y 226.11,Z 464.053,A -85,B 0,C 180,E1 -19882.858,E2 -19882.858} C_VEL
LIN {X 0,Y 226.077,Z 462.487,A -85,B 0,C 180,E1 -19885.169,E2 -19885.169} C_VEL
LIN {X 0,Y 225.887,Z 465.947,A -85,B 0,C 180,E1 -19888.217,E2 -19888.217} C_VEL
LIN {X 0,Y 225.883,Z 467.263,A -85,B 0,C 180,E1 -19890,E2 -19890} C_VEL
LIN {X 0,Y 225.839,Z 468.092,A -85,B 0,C 180,E1 -19891.783,E2 -19891.783} C_VEL
LIN {X 0,Y 225.731,Z 468.362,A -85,B 0,C 180,E1 -19893.57,E2 -19893.57} C_VEL
LIN {X 0,Y 225.78,Z 468.085,A -85,B 0,C 180,E1 -19895.358,E2 -19895.358} C_VEL
LIN {X 0,Y 225.934,Z 467.357,A -85,B 0,C 180,E1 -19897.147,E2 -19897.147} C_VEL
LIN {X 0,Y 226.294,Z 466.172,A -85,B 0,C 180,E1 -19898.933,E2 -19898.933} C_VEL
LIN {X 0,Y 227.228,Z 463.341,A -85,B 0,C 180,E1 -19901.597,E2 -19901.597} C_VEL
LIN {X 0,Y 228.684,Z 459.283,A -85,B 0,C 180,E1 -19904.232,E2 -19904.232} C_VEL
LIN {X 0,Y 230.628,Z 453.85,A -85,B 0,C 180,E1 -19906.827,E2 -19906.827} C_VEL
LIN {X 0,Y 233.136,Z 446.541,A -85,B 0,C 180,E1 -19909.366,E2 -19909.366} C_VEL
LIN {X 0,Y 235.185,Z 440.496,A -85,B 0,C 180,E1 -19911.014,E2 -19911.014} C_VEL
LIN {X 0,Y 237.129,Z 433.185,A -85,B 0,C 180,E1 -19912.662,E2 -19912.662} C_VEL
LIN {X 0,Y 239.396,Z 425.347,A -85,B 0,C 180,E1 -19914.037,E2 -19914.037} C_VEL
LIN {X 0,Y 240.9,Z 418.613,A -85,B 0,C 180,E1 -19915.025,E2 -19915.025} C_VEL
LIN {X 0,Y 242.624,Z 410.391,A -85,B 0,C 180,E1 -19915.984,E2 -19915.984} C_VEL
LIN {X 0,Y 244.121,Z 402.052,A -85,B 0,C 180,E1 -19916.732,E2 -19916.732} C_VEL
LIN {X 0,Y 245.341,Z 392.818,A -85,B 0,C 180,E1 -19917.355,E2 -19917.355} C_VEL
LIN {X 0,Y 246.18,Z 383.762,A -85,B 0,C 180,E1 -19917.766,E2 -19917.766} C_VEL
LIN {X 0,Y 247.079,Z 358.281,A -85,B 0,C 180,E1 -19918.563,E2 -19918.563} C_VEL
LIN {X 0,Y 244.062,Z 338.57,A -85,B 0,C 180,E1 -19919.753,E2 -19919.753} C_VEL
LIN {X 0,Y 241.736,Z 327.613,A -85,B 0,C 180,E1 -19920.55,E2 -19920.55} C_VEL
LIN {X 0,Y 235.351,Z 314.04,A -85,B 0,C 180,E1 -19922.229,E2 -19922.229} C_VEL
LIN {X 0,Y 231.495,Z 306.397,A -85,B 0,C 180,E1 -19923.288,E2 -19923.288} C_VEL
LIN {X 0,Y 231.278,Z 305.659,A -85,B 0,C 180,E1 -19923.492,E2 -19923.492} C_VEL
LIN {X 0,Y 229.632,Z 298.416,A -85,B 0,C 180,E1 -19927.268,E2 -19927.268} C_VEL
LIN {X 0,Y 227.866,Z 291.909,A -85,B 0,C 180,E1 -19931.097,E2 -19931.097} C_VEL
LIN {X 0,Y 227.831,Z 291.915,A -85,B 0,C 180,E1 -19935.193,E2 -19935.193} C_VEL
LIN {X 0,Y 227.808,Z 291.919,A -85,B 0,C 180,E1 -19939.614,E2 -19939.614} C_VEL
LIN {X 0,Y 227.873,Z 291.904,A -85,B 0,C 180,E1 -19944.121,E2 -19944.121} C_VEL
LIN {X 0,Y 227.865,Z 291.904,A -85,B 0,C 180,E1 -19948.372,E2 -19948.372} C_VEL
LIN {X 0,Y 227.864,Z 291.909,A -85,B 0,C 180,E1 -19952.437,E2 -19952.437} C_VEL
LIN {X 0,Y 227.902,Z 291.909,A -85,B 0,C 180,E1 -19956.361,E2 -19956.361} C_VEL
LIN {X 0,Y 227.932,Z 291.9,A -85,B 0,C 180,E1 -19960.168,E2 -19960.168} C_VEL
LIN {X 0,Y 228.035,Z 291.877,A -85,B 0,C 180,E1 -19963.891,E2 -19963.891} C_VEL
LIN {X 0,Y 228.072,Z 291.878,A -85,B 0,C 180,E1 -19967.538,E2 -19967.538} C_VEL
LIN {X 0,Y 228.271,Z 291.856,A -85,B 0,C 180,E1 -19971.139,E2 -19971.139} C_VEL
LIN {X 0,Y 228.326,Z 291.847,A -85,B 0,C 180,E1 -19972.922,E2 -19972.922} C_VEL
LIN {X 0,Y 228.55,Z 291.818,A -85,B 0,C 180,E1 -19978.232,E2 -19978.232} C_VEL
LIN {X 0,Y 228.55,Z 291.82,A -85,B 0,C 180,E1 -19981.756,E2 -19981.756} C_VEL
LIN {X 0,Y 228.308,Z 291.854,A -85,B 0,C 180,E1 -19987.067,E2 -19987.067} C_VEL
LIN {X 0,Y 228.141,Z 291.865,A -85,B 0,C 180,E1 -19990.645,E2 -19990.645} C_VEL
LIN {X 0,Y 228.059,Z 291.885,A -85,B 0,C 180,E1 -19994.266,E2 -19994.266} C_VEL
LIN {X 0,Y 227.996,Z 291.897,A -85,B 0,C 180,E1 -19997.947,E2 -19997.947} C_VEL
LIN {X 0,Y 227.921,Z 291.907,A -85,B 0,C 180,E1 -20002.323,E2 -20002.323} C_VEL
LIN {X 0,Y 227.93,Z 291.907,A -85,B 0,C 180,E1 -20006.596,E2 -20006.596} C_VEL
LIN {X 0,Y 227.883,Z 291.914,A -85,B 0,C 180,E1 -20010.285,E2 -20010.285} C_VEL
LIN {X 0,Y 227.863,Z 291.913,A -85,B 0,C 180,E1 -20013.715,E2 -20013.715} C_VEL
LIN {X 0,Y 227.851,Z 291.916,A -85,B 0,C 180,E1 -20018.081,E2 -20018.081} C_VEL
LIN {X 0,Y 227.913,Z 291.903,A -85,B 0,C 180,E1 -20019.033,E2 -20019.033} C_VEL
LIN {X 0,Y 228.913,Z 294.732,A -85,B 0,C 180,E1 -20019.381,E2 -20019.381} C_VEL
LIN {X 0,Y 230.813,Z 297.273,A -85,B 0,C 180,E1 -20019.882,E2 -20019.882} C_VEL
LIN {X 0,Y 238.108,Z 309.122,A -85,B 0,C 180,E1 -20021.775,E2 -20021.775} C_VEL
LIN {X 0,Y 242.997,Z 317.881,A -85,B 0,C 180,E1 -20022.985,E2 -20022.985} C_VEL
LIN {X 0,Y 248.312,Z 329.883,A -85,B 0,C 180,E1 -20024.307,E2 -20024.307} C_VEL
LIN {X 0,Y 246.822,Z 365.438,A -85,B 0,C 180,E1 -20025.376,E2 -20025.376} C_VEL
LIN {X 0,Y 246.083,Z 374.953,A -85,B 0,C 180,E1 -20025.856,E2 -20025.856} C_VEL
LIN {X 0,Y 244.93,Z 385.128,A -85,B 0,C 180,E1 -20026.618,E2 -20026.618} C_VEL
LIN {X 0,Y 243.138,Z 396.143,A -85,B 0,C 180,E1 -20027.775,E2 -20027.775} C_VEL
LIN {X 0,Y 241.183,Z 405.461,A -85,B 0,C 180,E1 -20029.1,E2 -20029.1} C_VEL
LIN {X 0,Y 239.464,Z 412.45,A -85,B 0,C 180,E1 -20030.332,E2 -20030.332} C_VEL
LIN {X 0,Y 237.81,Z 418.581,A -85,B 0,C 180,E1 -20031.639,E2 -20031.639} C_VEL
LIN {X 0,Y 235.7,Z 425.308,A -85,B 0,C 180,E1 -20033.391,E2 -20033.391} C_VEL
LIN {X 0,Y 233.775,Z 430.831,A -85,B 0,C 180,E1 -20035.167,E2 -20035.167} C_VEL
LIN {X 0,Y 232.092,Z 435.38,A -85,B 0,C 180,E1 -20036.972,E2 -20036.972} C_VEL
LIN {X 0,Y 230.681,Z 439.102,A -85,B 0,C 180,E1 -20038.807,E2 -20038.807} C_VEL
LIN {X 0,Y 228.872,Z 443.287,A -85,B 0,C 180,E1 -20041.578,E2 -20041.578} C_VEL
LIN {X 0,Y 227.477,Z 446.097,A -85,B 0,C 180,E1 -20044.372,E2 -20044.372} C_VEL
LIN {X 0,Y 226.76,Z 447.159,A -85,B 0,C 180,E1 -20046.24,E2 -20046.24} C_VEL
LIN {X 0,Y 226.098,Z 447.798,A -85,B 0,C 180,E1 -20048.809,E2 -20048.809} C_VEL
LIN {X 0,Y 225.646,Z 447.198,A -85,B 0,C 180,E1 -20051.853,E2 -20051.853} C_VEL
LIN {X 0,Y 225.595,Z 446.144,A -85,B 0,C 180,E1 -20053.718,E2 -20053.718} C_VEL
LIN {X 0,Y 225.772,Z 443.426,A -85,B 0,C 180,E1 -20056.499,E2 -20056.499} C_VEL
LIN {X 0,Y 226.053,Z 440.949,A -85,B 0,C 180,E1 -20058.341,E2 -20058.341} C_VEL
LIN {X 0,Y 226.421,Z 437.799,A -85,B 0,C 180,E1 -20060.171,E2 -20060.171} C_VEL
LIN {X 0,Y 227.197,Z 431.649,A -85,B 0,C 180,E1 -20062.893,E2 -20062.893} C_VEL
LIN {X 0,Y 227.735,Z 426.574,A -85,B 0,C 180,E1 -20064.688,E2 -20064.688} C_VEL
LIN {X 0,Y 228.61,Z 420.402,A -85,B 0,C 180,E1 -20066.475,E2 -20066.475} C_VEL
LIN {X 0,Y 229.567,Z 412.903,A -85,B 0,C 180,E1 -20068.246,E2 -20068.246} C_VEL
LIN {X 0,Y 230.556,Z 404.863,A -85,B 0,C 180,E1 -20069.782,E2 -20069.782} C_VEL
LIN {X 0,Y 231.752,Z 394.461,A -85,B 0,C 180,E1 -20071.347,E2 -20071.347} C_VEL
LIN {X 0,Y 232.645,Z 383.218,A -85,B 0,C 180,E1 -20072.568,E2 -20072.568} C_VEL
LIN {X 0,Y 233.217,Z 373.816,A -85,B 0,C 180,E1 -20073.307,E2 -20073.307} C_VEL
LIN {X 0,Y 233.617,Z 364.565,A -85,B 0,C 180,E1 -20073.802,E2 -20073.802} C_VEL
LIN {X 0,Y 234.74,Z 313.929,A -85,B 0,C 180,E1 -20075.387,E2 -20075.387} C_VEL
LIN {X 0,Y 233.284,Z 306.229,A -85,B 0,C 180,E1 -20075.745,E2 -20075.745} C_VEL
LIN {X 0,Y 228.29,Z 291.861,A -85,B 0,C 180,E1 -20076.63,E2 -20076.63} C_VEL
LIN {X 0,Y 228.113,Z 291.884,A -85,B 0,C 180,E1 -20080.653,E2 -20080.653} C_VEL
LIN {X 0,Y 228.015,Z 291.892,A -85,B 0,C 180,E1 -20086.106,E2 -20086.106} C_VEL
LIN {X 0,Y 227.908,Z 291.908,A -85,B 0,C 180,E1 -20089.829,E2 -20089.829} C_VEL
LIN {X 0,Y 227.868,Z 291.915,A -85,B 0,C 180,E1 -20093.638,E2 -20093.638} C_VEL
LIN {X 0,Y 227.828,Z 291.92,A -85,B 0,C 180,E1 -20097.563,E2 -20097.563} C_VEL
LIN {X 0,Y 227.831,Z 291.911,A -85,B 0,C 180,E1 -20101.629,E2 -20101.629} C_VEL
LIN {X 0,Y 227.842,Z 291.915,A -85,B 0,C 180,E1 -20105.879,E2 -20105.879} C_VEL
LIN {X 0,Y 227.785,Z 291.921,A -85,B 0,C 180,E1 -20110.386,E2 -20110.386} C_VEL
LIN {X 0,Y 227.804,Z 291.918,A -85,B 0,C 180,E1 -20115.201,E2 -20115.201} C_VEL
LIN {X 0,Y 227.808,Z 291.921,A -85,B 0,C 180,E1 -20119.629,E2 -20119.629} C_VEL
LIN {X 0,Y 227.866,Z 291.913,A -85,B 0,C 180,E1 -20124.134,E2 -20124.134} C_VEL
LIN {X 0,Y 227.843,Z 291.914,A -85,B 0,C 180,E1 -20128.382,E2 -20128.382} C_VEL
LIN {X 0,Y 227.844,Z 291.914,A -85,B 0,C 180,E1 -20132.447,E2 -20132.447} C_VEL
LIN {X 0,Y 227.886,Z 291.901,A -85,B 0,C 180,E1 -20136.371,E2 -20136.371} C_VEL
LIN {X 0,Y 227.988,Z 291.884,A -85,B 0,C 180,E1 -20140.185,E2 -20140.185} C_VEL
LIN {X 0,Y 228.235,Z 291.907,A -85,B 0,C 180,E1 -20142.15,E2 -20142.15} C_VEL
LIN {X 0,Y 230.219,Z 310.948,A -85,B 0,C 180,E1 -20143.154,E2 -20143.154} C_VEL
LIN {X 0,Y 228.839,Z 366.6,A -85,B 0,C 180,E1 -20146.18,E2 -20146.18} C_VEL
LIN {X 0,Y 228.429,Z 378.307,A -85,B 0,C 180,E1 -20147.118,E2 -20147.118} C_VEL
LIN {X 0,Y 227.989,Z 390.387,A -85,B 0,C 180,E1 -20148.448,E2 -20148.448} C_VEL
LIN {X 0,Y 227.491,Z 399.595,A -85,B 0,C 180,E1 -20149.774,E2 -20149.774} C_VEL
LIN {X 0,Y 227.041,Z 408.436,A -85,B 0,C 180,E1 -20151.349,E2 -20151.349} C_VEL
LIN {X 0,Y 226.58,Z 418.096,A -85,B 0,C 180,E1 -20153.486,E2 -20153.486} C_VEL
LIN {X 0,Y 226.313,Z 425.52,A -85,B 0,C 180,E1 -20155.553,E2 -20155.553} C_VEL
LIN {X 0,Y 226.108,Z 430.832,A -85,B 0,C 180,E1 -20157.334,E2 -20157.334} C_VEL
LIN {X 0,Y 225.928,Z 435.293,A -85,B 0,C 180,E1 -20159.115,E2 -20159.115} C_VEL
LIN {X 0,Y 225.971,Z 440.635,A -85,B 0,C 180,E1 -20161.788,E2 -20161.788} C_VEL
LIN {X 0,Y 226.465,Z 444.606,A -85,B 0,C 180,E1 -20164.455,E2 -20164.455} C_VEL
LIN {X 0,Y 227.249,Z 447.264,A -85,B 0,C 180,E1 -20167.111,E2 -20167.111} C_VEL
LIN {X 0,Y 227.936,Z 448.431,A -85,B 0,C 180,E1 -20168.874,E2 -20168.874} C_VEL
LIN {X 0,Y 229.576,Z 449.088,A -85,B 0,C 180,E1 -20171.506,E2 -20171.506} C_VEL
LIN {X 0,Y 231.693,Z 448.834,A -85,B 0,C 180,E1 -20174.049,E2 -20174.049} C_VEL
LIN {X 0,Y 234.184,Z 447.524,A -85,B 0,C 180,E1 -20176.295,E2 -20176.295} C_VEL
LIN {X 0,Y 235.235,Z 446.468,A -85,B 0,C 180,E1 -20177.691,E2 -20177.691} C_VEL
LIN {X 0,Y 235.651,Z 444.436,A -85,B 0,C 180,E1 -20180.058,E2 -20180.058} C_VEL
LIN {X 0,Y 236.432,Z 441.722,A -85,B 0,C 180,E1 -20182.35,E2 -20182.35} C_VEL
LIN {X 0,Y 237.996,Z 439.421,A -85,B 0,C 180,E1 -20183.599,E2 -20183.599} C_VEL
LIN {X 0,Y 242.478,Z 433.792,A -85,B 0,C 180,E1 -20185.775,E2 -20185.775} C_VEL
LIN {X 0,Y 247.551,Z 426.351,A -85,B 0,C 180,E1 -20187.938,E2 -20187.938} C_VEL
LIN {X 0,Y 252.084,Z 418.409,A -85,B 0,C 180,E1 -20189.665,E2 -20189.665} C_VEL
LIN {X 0,Y 256.896,Z 408.652,A -85,B 0,C 180,E1 -20191.323,E2 -20191.323} C_VEL
LIN {X 0,Y 260.959,Z 398.678,A -85,B 0,C 180,E1 -20192.595,E2 -20192.595} C_VEL
LIN {X 0,Y 264.044,Z 389.541,A -85,B 0,C 180,E1 -20193.529,E2 -20193.529} C_VEL
LIN {X 0,Y 267.417,Z 377.11,A -85,B 0,C 180,E1 -20194.473,E2 -20194.473} C_VEL
LIN {X 0,Y 270.155,Z 364.169,A -85,B 0,C 180,E1 -20195.148,E2 -20195.148} C_VEL
LIN {X 0,Y 271.197,Z 358.506,A -85,B 0,C 180,E1 -20195.448,E2 -20195.448} C_VEL
LIN {X 0,Y 269.502,Z 354.182,A -85,B 0,C 180,E1 -20197.353,E2 -20197.353} C_VEL
LIN {X 0,Y 268.155,Z 351.316,A -85,B 0,C 180,E1 -20199.213,E2 -20199.213} C_VEL
LIN {X 0,Y 267.046,Z 349.018,A -85,B 0,C 180,E1 -20201.53,E2 -20201.53} C_VEL
LIN {X 0,Y 266.505,Z 348.46,A -85,B 0,C 180,E1 -20203.291,E2 -20203.291} C_VEL
LIN {X 0,Y 266.662,Z 348.768,A -85,B 0,C 180,E1 -20206.745,E2 -20206.745} C_VEL
LIN {X 0,Y 267.016,Z 349.454,A -85,B 0,C 180,E1 -20207.84,E2 -20207.84} C_VEL
LIN {X 0,Y 268.698,Z 353.555,A -85,B 0,C 180,E1 -20211.116,E2 -20211.116} C_VEL
LIN {X 0,Y 269.896,Z 356.403,A -85,B 0,C 180,E1 -20212.597,E2 -20212.597} C_VEL
LIN {X 0,Y 270.561,Z 358.218,A -85,B 0,C 180,E1 -20213.389,E2 -20213.389} C_VEL
LIN {X 0,Y 269.608,Z 368.297,A -85,B 0,C 180,E1 -20214.434,E2 -20214.434} C_VEL
LIN {X 0,Y 265.742,Z 387.251,A -85,B 0,C 180,E1 -20215.433,E2 -20215.433} C_VEL
LIN {X 0,Y 262.462,Z 398.499,A -85,B 0,C 180,E1 -20216.2,E2 -20216.2} C_VEL
LIN {X 0,Y 258.748,Z 408.877,A -85,B 0,C 180,E1 -20217.096,E2 -20217.096} C_VEL
LIN {X 0,Y 254.198,Z 419.385,A -85,B 0,C 180,E1 -20218.311,E2 -20218.311} C_VEL
LIN {X 0,Y 249.918,Z 427.881,A -85,B 0,C 180,E1 -20219.59,E2 -20219.59} C_VEL
LIN {X 0,Y 244.998,Z 436.674,A -85,B 0,C 180,E1 -20221.282,E2 -20221.282} C_VEL
LIN {X 0,Y 240.492,Z 443.702,A -85,B 0,C 180,E1 -20223.066,E2 -20223.066} C_VEL
LIN {X 0,Y 236.344,Z 449.443,A -85,B 0,C 180,E1 -20224.929,E2 -20224.929} C_VEL
LIN {X 0,Y 232.633,Z 454.1,A -85,B 0,C 180,E1 -20226.875,E2 -20226.875} C_VEL
LIN {X 0,Y 228.803,Z 458.409,A -85,B 0,C 180,E1 -20229.314,E2 -20229.314} C_VEL
LIN {X 0,Y 225.388,Z 461.566,A -85,B 0,C 180,E1 -20231.831,E2 -20231.831} C_VEL
LIN {X 0,Y 223.666,Z 462.983,A -85,B 0,C 180,E1 -20233.572,E2 -20233.572} C_VEL
LIN {X 0,Y 222.194,Z 463.979,A -85,B 0,C 180,E1 -20235.342,E2 -20235.342} C_VEL
LIN {X 0,Y 220.998,Z 464.514,A -85,B 0,C 180,E1 -20237.137,E2 -20237.137} C_VEL
LIN {X 0,Y 220.087,Z 464.476,A -85,B 0,C 180,E1 -20238.954,E2 -20238.954} C_VEL
LIN {X 0,Y 219.437,Z 464.009,A -85,B 0,C 180,E1 -20240.785,E2 -20240.785} C_VEL
LIN {X 0,Y 219.114,Z 463.119,A -85,B 0,C 180,E1 -20242.628,E2 -20242.628} C_VEL
LIN {X 0,Y 219.064,Z 461.602,A -85,B 0,C 180,E1 -20244.779,E2 -20244.779} C_VEL
LIN {X 0,Y 218.822,Z 465.462,A -85,B 0,C 180,E1 -20248.159,E2 -20248.159} C_VEL
LIN {X 0,Y 218.815,Z 466.842,A -85,B 0,C 180,E1 -20250,E2 -20250} C_VEL
LIN {X 0,Y 218.768,Z 467.721,A -85,B 0,C 180,E1 -20251.841,E2 -20251.841} C_VEL
LIN {X 0,Y 218.637,Z 467.942,A -85,B 0,C 180,E1 -20254.763,E2 -20254.763} C_VEL
LIN {X 0,Y 218.871,Z 467.125,A -85,B 0,C 180,E1 -20257.379,E2 -20257.379} C_VEL
LIN {X 0,Y 219.262,Z 466.007,A -85,B 0,C 180,E1 -20259.222,E2 -20259.222} C_VEL
LIN {X 0,Y 220.264,Z 463.249,A -85,B 0,C 180,E1 -20261.969,E2 -20261.969} C_VEL
LIN {X 0,Y 221.791,Z 459.267,A -85,B 0,C 180,E1 -20264.684,E2 -20264.684} C_VEL
LIN {X 0,Y 223.068,Z 455.844,A -85,B 0,C 180,E1 -20266.472,E2 -20266.472} C_VEL
LIN {X 0,Y 225.107,Z 450.55,A -85,B 0,C 180,E1 -20268.663,E2 -20268.663} C_VEL
LIN {X 0,Y 226.961,Z 445.376,A -85,B 0,C 180,E1 -20270.387,E2 -20270.387} C_VEL
LIN {X 0,Y 229.113,Z 439.167,A -85,B 0,C 180,E1 -20272.071,E2 -20272.071} C_VEL
LIN {X 0,Y 230.959,Z 432.671,A -85,B 0,C 180,E1 -20273.54,E2 -20273.54} C_VEL
LIN {X 0,Y 233.189,Z 424.81,A -85,B 0,C 180,E1 -20274.957,E2 -20274.957} C_VEL
LIN {X 0,Y 235.108,Z 417.071,A -85,B 0,C 180,E1 -20276.074,E2 -20276.074} C_VEL
LIN {X 0,Y 237.017,Z 407.875,A -85,B 0,C 180,E1 -20277.122,E2 -20277.122} C_VEL
LIN {X 0,Y 239.075,Z 395.712,A -85,B 0,C 180,E1 -20278.095,E2 -20278.095} C_VEL
LIN {X 0,Y 240.087,Z 386.033,A -85,B 0,C 180,E1 -20278.609,E2 -20278.609} C_VEL
LIN {X 0,Y 241.254,Z 362.006,A -85,B 0,C 180,E1 -20279.369,E2 -20279.369} C_VEL
LIN {X 0,Y 240.946,Z 357.203,A -85,B 0,C 180,E1 -20279.596,E2 -20279.596} C_VEL
LIN {X 0,Y 238.039,Z 338.487,A -85,B 0,C 180,E1 -20280.797,E2 -20280.797} C_VEL
LIN {X 0,Y 236.306,Z 330.515,A -85,B 0,C 180,E1 -20281.415,E2 -20281.415} C_VEL
LIN {X 0,Y 230.203,Z 317.604,A -85,B 0,C 180,E1 -20283.095,E2 -20283.095} C_VEL
LIN {X 0,Y 226,Z 309.484,A -85,B 0,C 180,E1 -20284.304,E2 -20284.304} C_VEL
LIN {X 0,Y 224.086,Z 305.426,A -85,B 0,C 180,E1 -20284.932,E2 -20284.932} C_VEL
LIN {X 0,Y 222.352,Z 298.466,A -85,B 0,C 180,E1 -20288.814,E2 -20288.814} C_VEL
LIN {X 0,Y 220.798,Z 292.792,A -85,B 0,C 180,E1 -20292.308,E2 -20292.308} C_VEL
LIN {X 0,Y 220.758,Z 292.793,A -85,B 0,C 180,E1 -20297.073,E2 -20297.073} C_VEL
LIN {X 0,Y 220.79,Z 292.787,A -85,B 0,C 180,E1 -20300.454,E2 -20300.454} C_VEL
LIN {X 0,Y 220.835,Z 292.789,A -85,B 0,C 180,E1 -20302.789,E2 -20302.789} C_VEL
LIN {X 0,Y 220.821,Z 292.791,A -85,B 0,C 180,E1 -20307.239,E2 -20307.239} C_VEL
LIN {X 0,Y 220.813,Z 292.793,A -85,B 0,C 180,E1 -20311.478,E2 -20311.478} C_VEL
LIN {X 0,Y 220.855,Z 292.785,A -85,B 0,C 180,E1 -20315.558,E2 -20315.558} C_VEL
LIN {X 0,Y 220.886,Z 292.772,A -85,B 0,C 180,E1 -20319.508,E2 -20319.508} C_VEL
LIN {X 0,Y 220.997,Z 292.754,A -85,B 0,C 180,E1 -20323.363,E2 -20323.363} C_VEL
LIN {X 0,Y 221.009,Z 292.763,A -85,B 0,C 180,E1 -20327.133,E2 -20327.133} C_VEL
LIN {X 0,Y 221.209,Z 292.735,A -85,B 0,C 180,E1 -20330.854,E2 -20330.854} C_VEL
LIN {X 0,Y 221.262,Z 292.727,A -85,B 0,C 180,E1 -20332.695,E2 -20332.695} C_VEL
LIN {X 0,Y 221.508,Z 292.696,A -85,B 0,C 180,E1 -20338.176,E2 -20338.176} C_VEL
LIN {X 0,Y 221.508,Z 292.697,A -85,B 0,C 180,E1 -20341.812,E2 -20341.812} C_VEL
LIN {X 0,Y 221.244,Z 292.735,A -85,B 0,C 180,E1 -20347.294,E2 -20347.294} C_VEL
LIN {X 0,Y 221.063,Z 292.747,A -85,B 0,C 180,E1 -20350.99,E2 -20350.99} C_VEL
LIN {X 0,Y 220.99,Z 292.762,A -85,B 0,C 180,E1 -20354.733,E2 -20354.733} C_VEL
LIN {X 0,Y 220.914,Z 292.779,A -85,B 0,C 180,E1 -20358.543,E2 -20358.543} C_VEL
LIN {X 0,Y 220.886,Z 292.784,A -85,B 0,C 180,E1 -20362.677,E2 -20362.677} C_VEL
LIN {X 0,Y 220.871,Z 292.784,A -85,B 0,C 180,E1 -20367.008,E2 -20367.008} C_VEL
LIN {X 0,Y 220.824,Z 292.789,A -85,B 0,C 180,E1 -20370.762,E2 -20370.762} C_VEL
LIN {X 0,Y 220.787,Z 292.779,A -85,B 0,C 180,E1 -20374.949,E2 -20374.949} C_VEL
LIN {X 0,Y 220.827,Z 292.844,A -85,B 0,C 180,E1 -20377.483,E2 -20377.483} C_VEL
LIN {X 0,Y 221.721,Z 295.457,A -85,B 0,C 180,E1 -20377.807,E2 -20377.807} C_VEL
LIN {X 0,Y 223.933,Z 298.332,A -85,B 0,C 180,E1 -20378.438,E2 -20378.438} C_VEL
LIN {X 0,Y 232.107,Z 311.252,A -85,B 0,C 180,E1 -20380.706,E2 -20380.706} C_VEL
LIN {X 0,Y 238.027,Z 321.87,A -85,B 0,C 180,E1 -20382.246,E2 -20382.246} C_VEL
LIN {X 0,Y 242.455,Z 331.958,A -85,B 0,C 180,E1 -20383.409,E2 -20383.409} C_VEL
LIN {X 0,Y 240.939,Z 366.142,A -85,B 0,C 180,E1 -20384.463,E2 -20384.463} C_VEL
LIN {X 0,Y 240.123,Z 375.881,A -85,B 0,C 180,E1 -20384.972,E2 -20384.972} C_VEL
LIN {X 0,Y 238.626,Z 387.698,A -85,B 0,C 180,E1 -20385.909,E2 -20385.909} C_VEL
LIN {X 0,Y 236.937,Z 397.166,A -85,B 0,C 180,E1 -20386.983,E2 -20386.983} C_VEL
LIN {X 0,Y 235.03,Z 405.858,A -85,B 0,C 180,E1 -20388.252,E2 -20388.252} C_VEL
LIN {X 0,Y 233.123,Z 413.253,A -85,B 0,C 180,E1 -20389.597,E2 -20389.597} C_VEL
LIN {X 0,Y 231.373,Z 419.301,A -85,B 0,C 180,E1 -20390.929,E2 -20390.929} C_VEL
LIN {X 0,Y 229.172,Z 425.961,A -85,B 0,C 180,E1 -20392.723,E2 -20392.723} C_VEL
LIN {X 0,Y 227.164,Z 431.429,A -85,B 0,C 180,E1 -20394.544,E2 -20394.544} C_VEL
LIN {X 0,Y 225.401,Z 435.93,A -85,B 0,C 180,E1 -20396.397,E2 -20396.397} C_VEL
LIN {X 0,Y 223.562,Z 440.396,A -85,B 0,C 180,E1 -20398.755,E2 -20398.755} C_VEL
LIN {X 0,Y 222.282,Z 443.152,A -85,B 0,C 180,E1 -20400.655,E2 -20400.655} C_VEL
LIN {X 0,Y 221.03,Z 445.557,A -85,B 0,C 180,E1 -20402.894,E2 -20402.894} C_VEL
LIN {X 0,Y 219.919,Z 447.302,A -85,B 0,C 180,E1 -20405.453,E2 -20405.453} C_VEL
LIN {X 0,Y 219.072,Z 448.127,A -85,B 0,C 180,E1 -20408.467,E2 -20408.467} C_VEL
LIN {X 0,Y 218.601,Z 447.707,A -85,B 0,C 180,E1 -20411.247,E2 -20411.247} C_VEL
LIN {X 0,Y 218.512,Z 446.695,A -85,B 0,C 180,E1 -20413.174,E2 -20413.174} C_VEL
LIN {X 0,Y 218.633,Z 444.223,A -85,B 0,C 180,E1 -20416.05,E2 -20416.05} C_VEL
LIN {X 0,Y 219.058,Z 440.326,A -85,B 0,C 180,E1 -20418.902,E2 -20418.902} C_VEL
LIN {X 0,Y 219.703,Z 434.975,A -85,B 0,C 180,E1 -20421.746,E2 -20421.746} C_VEL
LIN {X 0,Y 220.429,Z 429.327,A -85,B 0,C 180,E1 -20424.053,E2 -20424.053} C_VEL
LIN {X 0,Y 221.388,Z 422.101,A -85,B 0,C 180,E1 -20426.36,E2 -20426.36} C_VEL
LIN {X 0,Y 222.362,Z 414.864,A -85,B 0,C 180,E1 -20428.189,E2 -20428.189} C_VEL
LIN {X 0,Y 223.365,Z 407.15,A -85,B 0,C 180,E1 -20429.775,E2 -20429.775} C_VEL
LIN {X 0,Y 224.358,Z 399.041,A -85,B 0,C 180,E1 -20431.122,E2 -20431.122} C_VEL
LIN {X 0,Y 225.217,Z 390.33,A -85,B 0,C 180,E1 -20432.276,E2 -20432.276} C_VEL
LIN {X 0,Y 225.941,Z 381.175,A -85,B 0,C 180,E1 -20433.211,E2 -20433.211} C_VEL
LIN {X 0,Y 226.576,Z 370.277,A -85,B 0,C 180,E1 -20434.012,E2 -20434.012} C_VEL
LIN {X 0,Y 227.021,Z 355.869,A -85,B 0,C 180,E1 -20434.595,E2 -20434.595} C_VEL
LIN {X 0,Y 227.985,Z 314.848,A -85,B 0,C 180,E1 -20435.878,E2 -20435.878} C_VEL
LIN {X 0,Y 226.807,Z 308.58,A -85,B 0,C 180,E1 -20436.179,E2 -20436.179} C_VEL
LIN {X 0,Y 221.238,Z 292.74,A -85,B 0,C 180,E1 -20437.198,E2 -20437.198} C_VEL
LIN {X 0,Y 221.033,Z 292.766,A -85,B 0,C 180,E1 -20440.998,E2 -20440.998} C_VEL
LIN {X 0,Y 220.979,Z 292.769,A -85,B 0,C 180,E1 -20446.633,E2 -20446.633} C_VEL
LIN {X 0,Y 220.858,Z 292.784,A -85,B 0,C 180,E1 -20450.49,E2 -20450.49} C_VEL
LIN {X 0,Y 220.821,Z 292.79,A -85,B 0,C 180,E1 -20454.441,E2 -20454.441} C_VEL
LIN {X 0,Y 220.777,Z 292.795,A -85,B 0,C 180,E1 -20458.522,E2 -20458.522} C_VEL
LIN {X 0,Y 220.787,Z 292.787,A -85,B 0,C 180,E1 -20462.761,E2 -20462.761} C_VEL
LIN {X 0,Y 220.779,Z 292.795,A -85,B 0,C 180,E1 -20467.28,E2 -20467.28} C_VEL
LIN {X 0,Y 220.737,Z 292.8,A -85,B 0,C 180,E1 -20471.961,E2 -20471.961} C_VEL
LIN {X 0,Y 220.747,Z 292.798,A -85,B 0,C 180,E1 -20475.549,E2 -20475.549} C_VEL
LIN {X 0,Y 220.79,Z 292.79,A -85,B 0,C 180,E1 -20480.469,E2 -20480.469} C_VEL
LIN {X 0,Y 220.787,Z 292.793,A -85,B 0,C 180,E1 -20485.051,E2 -20485.051} C_VEL
LIN {X 0,Y 220.822,Z 292.788,A -85,B 0,C 180,E1 -20489.396,E2 -20489.396} C_VEL
LIN {X 0,Y 220.866,Z 292.784,A -85,B 0,C 180,E1 -20493.553,E2 -20493.553} C_VEL
LIN {X 0,Y 220.86,Z 292.775,A -85,B 0,C 180,E1 -20497.559,E2 -20497.559} C_VEL
LIN {X 0,Y 221.198,Z 292.721,A -85,B 0,C 180,E1 -20502.183,E2 -20502.183} C_VEL
LIN {X 0,Y 223.094,Z 311.51,A -85,B 0,C 180,E1 -20503.209,E2 -20503.209} C_VEL
LIN {X 0,Y 221.768,Z 366.361,A -85,B 0,C 180,E1 -20506.315,E2 -20506.315} C_VEL
LIN {X 0,Y 221.382,Z 378.029,A -85,B 0,C 180,E1 -20507.283,E2 -20507.283} C_VEL
LIN {X 0,Y 220.962,Z 389.319,A -85,B 0,C 180,E1 -20508.54,E2 -20508.54} C_VEL
LIN {X 0,Y 220.413,Z 400.038,A -85,B 0,C 180,E1 -20510.138,E2 -20510.138} C_VEL
LIN {X 0,Y 219.982,Z 408.755,A -85,B 0,C 180,E1 -20511.741,E2 -20511.741} C_VEL
LIN {X 0,Y 219.518,Z 418.257,A -85,B 0,C 180,E1 -20513.901,E2 -20513.901} C_VEL
LIN {X 0,Y 219.289,Z 425.211,A -85,B 0,C 180,E1 -20515.871,E2 -20515.871} C_VEL
LIN {X 0,Y 219.068,Z 430.614,A -85,B 0,C 180,E1 -20517.708,E2 -20517.708} C_VEL
LIN {X 0,Y 218.874,Z 436.096,A -85,B 0,C 180,E1 -20520.006,E2 -20520.006} C_VEL
LIN {X 0,Y 219.037,Z 441.328,A -85,B 0,C 180,E1 -20522.764,E2 -20522.764} C_VEL
LIN {X 0,Y 219.681,Z 445.222,A -85,B 0,C 180,E1 -20525.513,E2 -20525.513} C_VEL
LIN {X 0,Y 220.205,Z 447.056,A -85,B 0,C 180,E1 -20527.34,E2 -20527.34} C_VEL
LIN {X 0,Y 220.935,Z 448.366,A -85,B 0,C 180,E1 -20529.157,E2 -20529.157} C_VEL
LIN {X 0,Y 221.917,Z 449.239,A -85,B 0,C 180,E1 -20530.959,E2 -20530.959} C_VEL
LIN {X 0,Y 223.713,Z 449.63,A -85,B 0,C 180,E1 -20533.124,E2 -20533.124} C_VEL
LIN {X 0,Y 224.856,Z 449.547,A -85,B 0,C 180,E1 -20534.486,E2 -20534.486} C_VEL
LIN {X 0,Y 227.502,Z 448.46,A -85,B 0,C 180,E1 -20536.823,E2 -20536.823} C_VEL
LIN {X 0,Y 231.1,Z 446.138,A -85,B 0,C 180,E1 -20539.549,E2 -20539.549} C_VEL
LIN {X 0,Y 235.013,Z 442.628,A -85,B 0,C 180,E1 -20541.956,E2 -20541.956} C_VEL
LIN {X 0,Y 237.996,Z 439.421,A -85,B 0,C 180,E1 -20543.599,E2 -20543.599} C_VEL
LIN {X 0,Y 239.697,Z 436.955,A -85,B 0,C 180,E1 -20544.819,E2 -20544.819} C_VEL
LIN {X 0,Y 241.267,Z 432.805,A -85,B 0,C 180,E1 -20546.944,E2 -20546.944} C_VEL
LIN {X 0,Y 243.071,Z 428.139,A -85,B 0,C 180,E1 -20548.942,E2 -20548.942} C_VEL
LIN {X 0,Y 245.052,Z 424.598,A -85,B 0,C 180,E1 -20549.944,E2 -20549.944} C_VEL
LIN {X 0,Y 250.402,Z 415.598,A -85,B 0,C 180,E1 -20551.757,E2 -20551.757} C_VEL
LIN {X 0,Y 255.031,Z 405.975,A -85,B 0,C 180,E1 -20553.214,E2 -20553.214} C_VEL
LIN {X 0,Y 259.369,Z 395.573,A -85,B 0,C 180,E1 -20554.451,E2 -20554.451} C_VEL
LIN {X 0,Y 262.88,Z 384.906,A -85,B 0,C 180,E1 -20555.387,E2 -20555.387} C_VEL
LIN {X 0,Y 265.448,Z 375.086,A -85,B 0,C 180,E1 -20556.053,E2 -20556.053} C_VEL
LIN {X 0,Y 268.036,Z 362.896,A -85,B 0,C 180,E1 -20556.672,E2 -20556.672} C_VEL
LIN {X 0,Y 266.785,Z 359.704,A -85,B 0,C 180,E1 -20558.331,E2 -20558.331} C_VEL
LIN {X 0,Y 266.087,Z 357.95,A -85,B 0,C 180,E1 -20559.52,E2 -20559.52} C_VEL
LIN {X 0,Y 265.003,Z 355.667,A -85,B 0,C 180,E1 -20562.048,E2 -20562.048} C_VEL
LIN {X 0,Y 264.559,Z 355.265,A -85,B 0,C 180,E1 -20564.171,E2 -20564.171} C_VEL
LIN {X 0,Y 264.925,Z 355.763,A -85,B 0,C 180,E1 -20567.146,E2 -20567.146} C_VEL
LIN {X 0,Y 266.437,Z 359.83,A -85,B 0,C 180,E1 -20570.586,E2 -20570.586} C_VEL
LIN {X 0,Y 267.59,Z 362.949,A -85,B 0,C 180,E1 -20572.234,E2 -20572.234} C_VEL
LIN {X 0,Y 267.645,Z 363.631,A -85,B 0,C 180,E1 -20572.407,E2 -20572.407} C_VEL
LIN {X 0,Y 266.758,Z 370.447,A -85,B 0,C 180,E1 -20573.1,E2 -20573.1} C_VEL
LIN {X 0,Y 263.053,Z 387.315,A -85,B 0,C 180,E1 -20574,E2 -20574} C_VEL
LIN {X 0,Y 259.729,Z 398.086,A -85,B 0,C 180,E1 -20574.727,E2 -20574.727} C_VEL
LIN {X 0,Y 255.409,Z 409.383,A -85,B 0,C 180,E1 -20575.702,E2 -20575.702} C_VEL
LIN {X 0,Y 250.122,Z 420.532,A -85,B 0,C 180,E1 -20577.016,E2 -20577.016} C_VEL
LIN {X 0,Y 245.126,Z 429.754,A -85,B 0,C 180,E1 -20578.449,E2 -20578.449} C_VEL
LIN {X 0,Y 239.973,Z 437.93,A -85,B 0,C 180,E1 -20580.14,E2 -20580.14} C_VEL
LIN {X 0,Y 235.227,Z 444.603,A -85,B 0,C 180,E1 -20581.928,E2 -20581.928} C_VEL
LIN {X 0,Y 230.861,Z 450.07,A -85,B 0,C 180,E1 -20583.805,E2 -20583.805} C_VEL
LIN {X 0,Y 226.205,Z 455.281,A -85,B 0,C 180,E1 -20586.177,E2 -20586.177} C_VEL
LIN {X 0,Y 222.229,Z 459.206,A -85,B 0,C 180,E1 -20588.673,E2 -20588.673} C_VEL
LIN {X 0,Y 218.662,Z 461.904,A -85,B 0,C 180,E1 -20591.251,E2 -20591.251} C_VEL
LIN {X 0,Y 216.858,Z 463.099,A -85,B 0,C 180,E1 -20593.041,E2 -20593.041} C_VEL
LIN {X 0,Y 215.335,Z 463.773,A -85,B 0,C 180,E1 -20594.864,E2 -20594.864} C_VEL
LIN {X 0,Y 214.103,Z 464.05,A -85,B 0,C 180,E1 -20596.716,E2 -20596.716} C_VEL
LIN {X 0,Y 213.148,Z 463.908,A -85,B 0,C 180,E1 -20598.589,E2 -20598.589} C_VEL
LIN {X 0,Y 212.47,Z 463.208,A -85,B 0,C 180,E1 -20600.48,E2 -20600.48} C_VEL
LIN {X 0,Y 212.104,Z 460.487,A -85,B 0,C 180,E1 -20604.295,E2 -20604.295} C_VEL
LIN {X 0,Y 211.784,Z 463.001,A -85,B 0,C 180,E1 -20606.194,E2 -20606.194} C_VEL
LIN {X 0,Y 211.758,Z 464.969,A -85,B 0,C 180,E1 -20608.098,E2 -20608.098} C_VEL
LIN {X 0,Y 211.748,Z 466.416,A -85,B 0,C 180,E1 -20610,E2 -20610} C_VEL
LIN {X 0,Y 211.675,Z 467.326,A -85,B 0,C 180,E1 -20611.902,E2 -20611.902} C_VEL
LIN {X 0,Y 211.55,Z 467.694,A -85,B 0,C 180,E1 -20614.645,E2 -20614.645} C_VEL
LIN {X 0,Y 211.832,Z 466.895,A -85,B 0,C 180,E1 -20617.626,E2 -20617.626} C_VEL
LIN {X 0,Y 212.249,Z 465.834,A -85,B 0,C 180,E1 -20619.529,E2 -20619.529} C_VEL
LIN {X 0,Y 213.318,Z 463.157,A -85,B 0,C 180,E1 -20622.365,E2 -20622.365} C_VEL
LIN {X 0,Y 214.357,Z 460.769,A -85,B 0,C 180,E1 -20624.235,E2 -20624.235} C_VEL
LIN {X 0,Y 216.263,Z 455.909,A -85,B 0,C 180,E1 -20627.006,E2 -20627.006} C_VEL
LIN {X 0,Y 218.407,Z 450.703,A -85,B 0,C 180,E1 -20629.258,E2 -20629.258} C_VEL
LIN {X 0,Y 220.88,Z 444.209,A -85,B 0,C 180,E1 -20631.463,E2 -20631.463} C_VEL
LIN {X 0,Y 223.117,Z 437.843,A -85,B 0,C 180,E1 -20633.187,E2 -20633.187} C_VEL
LIN {X 0,Y 225.193,Z 431.149,A -85,B 0,C 180,E1 -20634.671,E2 -20634.671} C_VEL
LIN {X 0,Y 227.994,Z 421.259,A -85,B 0,C 180,E1 -20636.407,E2 -20636.407} C_VEL
LIN {X 0,Y 230.413,Z 410.976,A -85,B 0,C 180,E1 -20637.72,E2 -20637.72} C_VEL
LIN {X 0,Y 232.201,Z 401.81,A -85,B 0,C 180,E1 -20638.593,E2 -20638.593} C_VEL
LIN {X 0,Y 233.532,Z 392.716,A -85,B 0,C 180,E1 -20639.235,E2 -20639.235} C_VEL
LIN {X 0,Y 234.465,Z 383.379,A -85,B 0,C 180,E1 -20639.685,E2 -20639.685} C_VEL
LIN {X 0,Y 235.424,Z 360.339,A -85,B 0,C 180,E1 -20640.438,E2 -20640.438} C_VEL
LIN {X 0,Y 232.59,Z 341.171,A -85,B 0,C 180,E1 -20641.697,E2 -20641.697} C_VEL
LIN {X 0,Y 231.117,Z 333.988,A -85,B 0,C 180,E1 -20642.261,E2 -20642.261} C_VEL
LIN {X 0,Y 225.309,Z 321.434,A -85,B 0,C 180,E1 -20643.955,E2 -20643.955} C_VEL
LIN {X 0,Y 220.92,Z 312.961,A -85,B 0,C 180,E1 -20645.288,E2 -20645.288} C_VEL
LIN {X 0,Y 219.04,Z 309.385,A -85,B 0,C 180,E1 -20645.882,E2 -20645.882} C_VEL
LIN {X 0,Y 216.81,Z 304.977,A -85,B 0,C 180,E1 -20646.639,E2 -20646.639} C_VEL
LIN {X 0,Y 214.77,Z 297.471,A -85,B 0,C 180,E1 -20651.174,E2 -20651.174} C_VEL
LIN {X 0,Y 213.714,Z 293.672,A -85,B 0,C 180,E1 -20653.676,E2 -20653.676} C_VEL
LIN {X 0,Y 213.713,Z 293.675,A -85,B 0,C 180,E1 -20656.342,E2 -20656.342} C_VEL
LIN {X 0,Y 213.713,Z 293.668,A -85,B 0,C 180,E1 -20661.325,E2 -20661.325} C_VEL
LIN {X 0,Y 213.763,Z 293.664,A -85,B 0,C 180,E1 -20666.013,E2 -20666.013} C_VEL
LIN {X 0,Y 213.759,Z 293.666,A -85,B 0,C 180,E1 -20670.445,E2 -20670.445} C_VEL
LIN {X 0,Y 213.789,Z 293.659,A -85,B 0,C 180,E1 -20674.694,E2 -20674.694} C_VEL
LIN {X 0,Y 213.807,Z 293.65,A -85,B 0,C 180,E1 -20678.797,E2 -20678.797} C_VEL
LIN {X 0,Y 213.927,Z 293.638,A -85,B 0,C 180,E1 -20682.797,E2 -20682.797} C_VEL
LIN {X 0,Y 213.949,Z 293.642,A -85,B 0,C 180,E1 -20686.701,E2 -20686.701} C_VEL
LIN {X 0,Y 214.146,Z 293.61,A -85,B 0,C 180,E1 -20690.55,E2 -20690.55} C_VEL
LIN {X 0,Y 214.095,Z 293.608,A -85,B 0,C 180,E1 -20694.343,E2 -20694.343} C_VEL
LIN {X 0,Y 214.441,Z 293.576,A -85,B 0,C 180,E1 -20698.116,E2 -20698.116} C_VEL
LIN {X 0,Y 214.542,Z 293.553,A -85,B 0,C 180,E1 -20699.994,E2 -20699.994} C_VEL
LIN {X 0,Y 214.441,Z 293.578,A -85,B 0,C 180,E1 -20701.872,E2 -20701.872} C_VEL
LIN {X 0,Y 214.185,Z 293.614,A -85,B 0,C 180,E1 -20707.536,E2 -20707.536} C_VEL
LIN {X 0,Y 213.994,Z 293.629,A -85,B 0,C 180,E1 -20711.358,E2 -20711.358} C_VEL
LIN {X 0,Y 213.927,Z 293.638,A -85,B 0,C 180,E1 -20715.231,E2 -20715.231} C_VEL
LIN {X 0,Y 213.832,Z 293.657,A -85,B 0,C 180,E1 -20719.181,E2 -20719.181} C_VEL
LIN {X 0,Y 213.837,Z 293.66,A -85,B 0,C 180,E1 -20723.221,E2 -20723.221} C_VEL
LIN {X 0,Y 213.817,Z 293.66,A -85,B 0,C 180,E1 -20727.444,E2 -20727.444} C_VEL
LIN {X 0,Y 213.753,Z 293.666,A -85,B 0,C 180,E1 -20731.732,E2 -20731.732} C_VEL
LIN {X 0,Y 213.719,Z 293.655,A -85,B 0,C 180,E1 -20735.739,E2 -20735.739} C_VEL
LIN {X 0,Y 214.616,Z 296.305,A -85,B 0,C 180,E1 -20736.108,E2 -20736.108} C_VEL
LIN {X 0,Y 216.898,Z 299.158,A -85,B 0,C 180,E1 -20736.812,E2 -20736.812} C_VEL
LIN {X 0,Y 219.199,Z 302.555,A -85,B 0,C 180,E1 -20737.521,E2 -20737.521} C_VEL
LIN {X 0,Y 227.321,Z 315.445,A -85,B 0,C 180,E1 -20739.896,E2 -20739.896} C_VEL
LIN {X 0,Y 233.233,Z 326.16,A -85,B 0,C 180,E1 -20741.514,E2 -20741.514} C_VEL
LIN {X 0,Y 236.723,Z 334.178,A -85,B 0,C 180,E1 -20742.476,E2 -20742.476} C_VEL
LIN {X 0,Y 235.119,Z 367.03,A -85,B 0,C 180,E1 -20743.505,E2 -20743.505} C_VEL
LIN {X 0,Y 234.183,Z 377.46,A -85,B 0,C 180,E1 -20744.08,E2 -20744.08} C_VEL
LIN {X 0,Y 232.548,Z 388.991,A -85,B 0,C 180,E1 -20745.055,E2 -20745.055} C_VEL
LIN {X 0,Y 230.799,Z 398.255,A -85,B 0,C 180,E1 -20746.152,E2 -20746.152} C_VEL
LIN {X 0,Y 229.082,Z 405.682,A -85,B 0,C 180,E1 -20747.253,E2 -20747.253} C_VEL
LIN {X 0,Y 227.133,Z 413.009,A -85,B 0,C 180,E1 -20748.594,E2 -20748.594} C_VEL
LIN {X 0,Y 224.984,Z 420.042,A -85,B 0,C 180,E1 -20750.181,E2 -20750.181} C_VEL
LIN {X 0,Y 223.033,Z 425.685,A -85,B 0,C 180,E1 -20751.723,E2 -20751.723} C_VEL
LIN {X 0,Y 221.106,Z 430.808,A -85,B 0,C 180,E1 -20753.418,E2 -20753.418} C_VEL
LIN {X 0,Y 219.17,Z 435.479,A -85,B 0,C 180,E1 -20755.307,E2 -20755.307} C_VEL
LIN {X 0,Y 217.636,Z 439.069,A -85,B 0,C 180,E1 -20757.084,E2 -20757.084} C_VEL
LIN {X 0,Y 215.749,Z 443.017,A -85,B 0,C 180,E1 -20759.675,E2 -20759.675} C_VEL
LIN {X 0,Y 214.041,Z 446.111,A -85,B 0,C 180,E1 -20762.633,E2 -20762.633} C_VEL
LIN {X 0,Y 213.118,Z 447.444,A -85,B 0,C 180,E1 -20764.615,E2 -20764.615} C_VEL
LIN {X 0,Y 212.446,Z 448.236,A -85,B 0,C 180,E1 -20766.611,E2 -20766.611} C_VEL
LIN {X 0,Y 211.961,Z 448.492,A -85,B 0,C 180,E1 -20768.61,E2 -20768.61} C_VEL
LIN {X 0,Y 211.583,Z 448.137,A -85,B 0,C 180,E1 -20770.6,E2 -20770.6} C_VEL
LIN {X 0,Y 211.427,Z 447.229,A -85,B 0,C 180,E1 -20772.593,E2 -20772.593} C_VEL
LIN {X 0,Y 211.462,Z 445.796,A -85,B 0,C 180,E1 -20774.581,E2 -20774.581} C_VEL
LIN {X 0,Y 211.717,Z 442.619,A -85,B 0,C 180,E1 -20777.54,E2 -20777.54} C_VEL
LIN {X 0,Y 212.292,Z 438.071,A -85,B 0,C 180,E1 -20780.473,E2 -20780.473} C_VEL
LIN {X 0,Y 212.961,Z 432.985,A -85,B 0,C 180,E1 -20782.891,E2 -20782.891} C_VEL
LIN {X 0,Y 213.744,Z 426.593,A -85,B 0,C 180,E1 -20785.285,E2 -20785.285} C_VEL
LIN {X 0,Y 214.671,Z 420.299,A -85,B 0,C 180,E1 -20787.186,E2 -20787.186} C_VEL
LIN {X 0,Y 215.573,Z 413.69,A -85,B 0,C 180,E1 -20788.833,E2 -20788.833} C_VEL
LIN {X 0,Y 216.653,Z 405.668,A -85,B 0,C 180,E1 -20790.465,E2 -20790.465} C_VEL
LIN {X 0,Y 217.863,Z 395.801,A -85,B 0,C 180,E1 -20792.056,E2 -20792.056} C_VEL
LIN {X 0,Y 218.876,Z 384.596,A -85,B 0,C 180,E1 -20793.379,E2 -20793.379} C_VEL
LIN {X 0,Y 219.532,Z 374.496,A -85,B 0,C 180,E1 -20794.229,E2 -20794.229} C_VEL
LIN {X 0,Y 219.976,Z 364.731,A -85,B 0,C 180,E1 -20794.777,E2 -20794.777} C_VEL
LIN {X 0,Y 221.261,Z 315.964,A -85,B 0,C 180,E1 -20796.384,E2 -20796.384} C_VEL
LIN {X 0,Y 220.051,Z 310.061,A -85,B 0,C 180,E1 -20796.689,E2 -20796.689} C_VEL
LIN {X 0,Y 214.169,Z 293.753,A -85,B 0,C 180,E1 -20797.78,E2 -20797.78} C_VEL
LIN {X 0,Y 213.965,Z 293.643,A -85,B 0,C 180,E1 -20801.367,E2 -20801.367} C_VEL
LIN {X 0,Y 213.889,Z 293.656,A -85,B 0,C 180,E1 -20805.241,E2 -20805.241} C_VEL
LIN {X 0,Y 213.808,Z 293.666,A -85,B 0,C 180,E1 -20809.191,E2 -20809.191} C_VEL
LIN {X 0,Y 213.776,Z 293.67,A -85,B 0,C 180,E1 -20813.236,E2 -20813.236} C_VEL
LIN {X 0,Y 213.761,Z 293.673,A -85,B 0,C 180,E1 -20817.431,E2 -20817.431} C_VEL
LIN {X 0,Y 213.734,Z 293.666,A -85,B 0,C 180,E1 -20821.744,E2 -20821.744} C_VEL
LIN {X 0,Y 213.718,Z 293.673,A -85,B 0,C 180,E1 -20826.294,E2 -20826.294} C_VEL
LIN {X 0,Y 213.681,Z 293.678,A -85,B 0,C 180,E1 -20831.133,E2 -20831.133} C_VEL
LIN {X 0,Y 213.683,Z 293.678,A -85,B 0,C 180,E1 -20833.685,E2 -20833.685} C_VEL
LIN {X 0,Y 213.685,Z 293.678,A -85,B 0,C 180,E1 -20836.351,E2 -20836.351} C_VEL
LIN {X 0,Y 213.699,Z 293.676,A -85,B 0,C 180,E1 -20839.149,E2 -20839.149} C_VEL
LIN {X 0,Y 213.729,Z 293.675,A -85,B 0,C 180,E1 -20843.718,E2 -20843.718} C_VEL
LIN {X 0,Y 213.746,Z 293.67,A -85,B 0,C 180,E1 -20848.267,E2 -20848.267} C_VEL
LIN {X 0,Y 213.778,Z 293.666,A -85,B 0,C 180,E1 -20852.604,E2 -20852.604} C_VEL
LIN {X 0,Y 213.803,Z 293.652,A -85,B 0,C 180,E1 -20856.986,E2 -20856.986} C_VEL
LIN {X 0,Y 214.162,Z 293.597,A -85,B 0,C 180,E1 -20862.231,E2 -20862.231} C_VEL
LIN {X 0,Y 215.995,Z 311.913,A -85,B 0,C 180,E1 -20863.283,E2 -20863.283} C_VEL
LIN {X 0,Y 214.672,Z 367.017,A -85,B 0,C 180,E1 -20866.578,E2 -20866.578} C_VEL
LIN {X 0,Y 214.348,Z 378.635,A -85,B 0,C 180,E1 -20867.581,E2 -20867.581} C_VEL
LIN {X 0,Y 213.885,Z 389.801,A -85,B 0,C 180,E1 -20868.876,E2 -20868.876} C_VEL
LIN {X 0,Y 213.359,Z 400.491,A -85,B 0,C 180,E1 -20870.527,E2 -20870.527} C_VEL
LIN {X 0,Y 212.86,Z 410.333,A -85,B 0,C 180,E1 -20872.417,E2 -20872.417} C_VEL
LIN {X 0,Y 212.48,Z 418.233,A -85,B 0,C 180,E1 -20874.312,E2 -20874.312} C_VEL
LIN {X 0,Y 212.268,Z 426.181,A -85,B 0,C 180,E1 -20876.685,E2 -20876.685} C_VEL
LIN {X 0,Y 211.929,Z 432.595,A -85,B 0,C 180,E1 -20879.056,E2 -20879.056} C_VEL
LIN {X 0,Y 211.898,Z 438.785,A -85,B 0,C 180,E1 -20881.907,E2 -20881.907} C_VEL
LIN {X 0,Y 212.383,Z 443.365,A -85,B 0,C 180,E1 -20884.751,E2 -20884.751} C_VEL
LIN {X 0,Y 213.187,Z 446.669,A -85,B 0,C 180,E1 -20887.583,E2 -20887.583} C_VEL
LIN {X 0,Y 214.651,Z 449.138,A -85,B 0,C 180,E1 -20890.81,E2 -20890.81} C_VEL
LIN {X 0,Y 216.51,Z 449.982,A -85,B 0,C 180,E1 -20893.139,E2 -20893.139} C_VEL
LIN {X 0,Y 218.018,Z 450.071,A -85,B 0,C 180,E1 -20894.95,E2 -20894.95} C_VEL
LIN {X 0,Y 220.036,Z 449.703,A -85,B 0,C 180,E1 -20896.712,E2 -20896.712} C_VEL
LIN {X 0,Y 222.177,Z 448.88,A -85,B 0,C 180,E1 -20898.446,E2 -20898.446} C_VEL
LIN {X 0,Y 224.848,Z 447.345,A -85,B 0,C 180,E1 -20900.33,E2 -20900.33} C_VEL
LIN {X 0,Y 228.633,Z 444.488,A -85,B 0,C 180,E1 -20902.602,E2 -20902.602} C_VEL
LIN {X 0,Y 233.152,Z 440.101,A -85,B 0,C 180,E1 -20904.967,E2 -20904.967} C_VEL
LIN {X 0,Y 238.396,Z 434.07,A -85,B 0,C 180,E1 -20907.333,E2 -20907.333} C_VEL
LIN {X 0,Y 243.522,Z 426.965,A -85,B 0,C 180,E1 -20909.386,E2 -20909.386} C_VEL
LIN {X 0,Y 245.052,Z 424.598,A -85,B 0,C 180,E1 -20909.944,E2 -20909.944} C_VEL
LIN {X 0,Y 247.103,Z 420.924,A -85,B 0,C 180,E1 -20910.91,E2 -20910.91} C_VEL
LIN {X 0,Y 249.295,Z 414.972,A -85,B 0,C 180,E1 -20912.678,E2 -20912.678} C_VEL
LIN {X 0,Y 251.543,Z 408.539,A -85,B 0,C 180,E1 -20914.299,E2 -20914.299} C_VEL
LIN {X 0,Y 253.424,Z 404.07,A -85,B 0,C 180,E1 -20915.039,E2 -20915.039} C_VEL
LIN {X 0,Y 257.615,Z 393.836,A -85,B 0,C 180,E1 -20916.158,E2 -20916.158} C_VEL
LIN {X 0,Y 261.222,Z 383.175,A -85,B 0,C 180,E1 -20917.039,E2 -20917.039} C_VEL
LIN {X 0,Y 264.648,Z 369.887,A -85,B 0,C 180,E1 -20917.816,E2 -20917.816} C_VEL
LIN {X 0,Y 265.134,Z 367.625,A -85,B 0,C 180,E1 -20917.919,E2 -20917.919} C_VEL
LIN {X 0,Y 264.106,Z 364.724,A -85,B 0,C 180,E1 -20919.696,E2 -20919.696} C_VEL
LIN {X 0,Y 263.135,Z 362.485,A -85,B 0,C 180,E1 -20922.127,E2 -20922.127} C_VEL
LIN {X 0,Y 262.732,Z 362.123,A -85,B 0,C 180,E1 -20924.071,E2 -20924.071} C_VEL
LIN {X 0,Y 263.036,Z 362.562,A -85,B 0,C 180,E1 -20926.995,E2 -20926.995} C_VEL
LIN {X 0,Y 264.329,Z 366.482,A -85,B 0,C 180,E1 -20930.29,E2 -20930.29} C_VEL
LIN {X 0,Y 264.903,Z 368.279,A -85,B 0,C 180,E1 -20931.314,E2 -20931.314} C_VEL
LIN {X 0,Y 264.238,Z 372.685,A -85,B 0,C 180,E1 -20931.737,E2 -20931.737} C_VEL
LIN {X 0,Y 260.375,Z 388.484,A -85,B 0,C 180,E1 -20932.585,E2 -20932.585} C_VEL
LIN {X 0,Y 256.366,Z 400.277,A -85,B 0,C 180,E1 -20933.398,E2 -20933.398} C_VEL
LIN {X 0,Y 251.614,Z 411.377,A -85,B 0,C 180,E1 -20934.405,E2 -20934.405} C_VEL
LIN {X 0,Y 246.84,Z 420.808,A -85,B 0,C 180,E1 -20935.536,E2 -20935.536} C_VEL
LIN {X 0,Y 241.555,Z 429.825,A -85,B 0,C 180,E1 -20936.939,E2 -20936.939} C_VEL
LIN {X 0,Y 236.118,Z 437.847,A -85,B 0,C 180,E1 -20938.608,E2 -20938.608} C_VEL
LIN {X 0,Y 231.048,Z 444.418,A -85,B 0,C 180,E1 -20940.377,E2 -20940.377} C_VEL
LIN {X 0,Y 226.37,Z 449.787,A -85,B 0,C 180,E1 -20942.244,E2 -20942.244} C_VEL
LIN {X 0,Y 222.957,Z 453.362,A -85,B 0,C 180,E1 -20943.812,E2 -20943.812} C_VEL
LIN {X 0,Y 218.372,Z 457.585,A -85,B 0,C 180,E1 -20946.278,E2 -20946.278} C_VEL
LIN {X 0,Y 214.356,Z 460.661,A -85,B 0,C 180,E1 -20948.859,E2 -20948.859} C_VEL
LIN {X 0,Y 211.955,Z 462.049,A -85,B 0,C 180,E1 -20950.635,E2 -20950.635} C_VEL
LIN {X 0,Y 210.068,Z 463.018,A -85,B 0,C 180,E1 -20952.476,E2 -20952.476} C_VEL
LIN {X 0,Y 208.497,Z 463.555,A -85,B 0,C 180,E1 -20954.355,E2 -20954.355} C_VEL
LIN {X 0,Y 207.225,Z 463.532,A -85,B 0,C 180,E1 -20956.266,E2 -20956.266} C_VEL
LIN {X 0,Y 205.515,Z 462.27,A -85,B 0,C 180,E1 -20960.154,E2 -20960.154} C_VEL
LIN {X 0,Y 205.194,Z 460.944,A -85,B 0,C 180,E1 -20962.125,E2 -20962.125} C_VEL
LIN {X 0,Y 205.171,Z 459.382,A -85,B 0,C 180,E1 -20963.796,E2 -20963.796} C_VEL
LIN {X 0,Y 204.723,Z 462.436,A -85,B 0,C 180,E1 -20966.063,E2 -20966.063} C_VEL
LIN {X 0,Y 204.672,Z 464.475,A -85,B 0,C 180,E1 -20968.032,E2 -20968.032} C_VEL
LIN {X 0,Y 204.682,Z 465.989,A -85,B 0,C 180,E1 -20970,E2 -20970} C_VEL
LIN {X 0,Y 204.585,Z 466.91,A -85,B 0,C 180,E1 -20971.968,E2 -20971.968} C_VEL
LIN {X 0,Y 204.481,Z 467.362,A -85,B 0,C 180,E1 -20974.584,E2 -20974.584} C_VEL
LIN {X 0,Y 204.77,Z 466.665,A -85,B 0,C 180,E1 -20977.89,E2 -20977.89} C_VEL
LIN {X 0,Y 205.229,Z 465.638,A -85,B 0,C 180,E1 -20979.859,E2 -20979.859} C_VEL
LIN {X 0,Y 206.39,Z 463.066,A -85,B 0,C 180,E1 -20982.787,E2 -20982.787} C_VEL
LIN {X 0,Y 208.05,Z 459.238,A -85,B 0,C 180,E1 -20985.678,E2 -20985.678} C_VEL
LIN {X 0,Y 210.335,Z 454.061,A -85,B 0,C 180,E1 -20988.507,E2 -20988.507} C_VEL
LIN {X 0,Y 212.693,Z 448.523,A -85,B 0,C 180,E1 -20990.806,E2 -20990.806} C_VEL
LIN {X 0,Y 215.527,Z 441.612,A -85,B 0,C 180,E1 -20993.035,E2 -20993.035} C_VEL
LIN {X 0,Y 218.08,Z 433.741,A -85,B 0,C 180,E1 -20995.022,E2 -20995.022} C_VEL
LIN {X 0,Y 220.469,Z 426.238,A -85,B 0,C 180,E1 -20996.505,E2 -20996.505} C_VEL
LIN {X 0,Y 222.587,Z 418.761,A -85,B 0,C 180,E1 -20997.696,E2 -20997.696} C_VEL
LIN {X 0,Y 224.578,Z 410.402,A -85,B 0,C 180,E1 -20998.759,E2 -20998.759} C_VEL
LIN {X 0,Y 226.261,Z 402.256,A -85,B 0,C 180,E1 -20999.555,E2 -20999.555} C_VEL
LIN {X 0,Y 227.719,Z 392.801,A -85,B 0,C 180,E1 -21000.246,E2 -21000.246} C_VEL
LIN {X 0,Y 228.716,Z 383.327,A -85,B 0,C 180,E1 -21000.717,E2 -21000.717} C_VEL
LIN {X 0,Y 229.744,Z 361.701,A -85,B 0,C 180,E1 -21001.431,E2 -21001.431} C_VEL
LIN {X 0,Y 226.997,Z 342.786,A -85,B 0,C 180,E1 -21002.723,E2 -21002.723} C_VEL
LIN {X 0,Y 225.788,Z 337.009,A -85,B 0,C 180,E1 -21003.206,E2 -21003.206} C_VEL
LIN {X 0,Y 220.595,Z 325.539,A -85,B 0,C 180,E1 -21004.82,E2 -21004.82} C_VEL
LIN {X 0,Y 214.862,Z 314.287,A -85,B 0,C 180,E1 -21006.676,E2 -21006.676} C_VEL
LIN {X 0,Y 211.84,Z 308.96,A -85,B 0,C 180,E1 -21007.689,E2 -21007.689} C_VEL
LIN {X 0,Y 209.524,Z 304.792,A -85,B 0,C 180,E1 -21008.503,E2 -21008.503} C_VEL
LIN {X 0,Y 207.489,Z 297.522,A -85,B 0,C 180,E1 -21013.101,E2 -21013.101} C_VEL
LIN {X 0,Y 206.615,Z 294.558,A -85,B 0,C 180,E1 -21015.242,E2 -21015.242} C_VEL
LIN {X 0,Y 206.656,Z 294.552,A -85,B 0,C 180,E1 -21019.741,E2 -21019.741} C_VEL
LIN {X 0,Y 206.709,Z 294.538,A -85,B 0,C 180,E1 -21024.685,E2 -21024.685} C_VEL
LIN {X 0,Y 206.704,Z 294.538,A -85,B 0,C 180,E1 -21029.33,E2 -21029.33} C_VEL
LIN {X 0,Y 206.713,Z 294.536,A -85,B 0,C 180,E1 -21033.763,E2 -21033.763} C_VEL
LIN {X 0,Y 206.74,Z 294.531,A -85,B 0,C 180,E1 -21038.035,E2 -21038.035} C_VEL
LIN {X 0,Y 206.874,Z 294.521,A -85,B 0,C 180,E1 -21042.191,E2 -21042.191} C_VEL
LIN {X 0,Y 206.889,Z 294.523,A -85,B 0,C 180,E1 -21046.238,E2 -21046.238} C_VEL
LIN {X 0,Y 207.103,Z 294.484,A -85,B 0,C 180,E1 -21050.225,E2 -21050.225} C_VEL
LIN {X 0,Y 207.057,Z 294.485,A -85,B 0,C 180,E1 -21054.15,E2 -21054.15} C_VEL
LIN {X 0,Y 207.377,Z 294.456,A -85,B 0,C 180,E1 -21058.052,E2 -21058.052} C_VEL
LIN {X 0,Y 207.508,Z 294.429,A -85,B 0,C 180,E1 -21059.994,E2 -21059.994} C_VEL
LIN {X 0,Y 207.377,Z 294.458,A -85,B 0,C 180,E1 -21061.936,E2 -21061.936} C_VEL
LIN {X 0,Y 207.129,Z 294.494,A -85,B 0,C 180,E1 -21067.794,E2 -21067.794} C_VEL
LIN {X 0,Y 206.92,Z 294.513,A -85,B 0,C 180,E1 -21071.752,E2 -21071.752} C_VEL
LIN {X 0,Y 206.86,Z 294.517,A -85,B 0,C 180,E1 -21075.764,E2 -21075.764} C_VEL
LIN {X 0,Y 206.778,Z 294.53,A -85,B 0,C 180,E1 -21079.862,E2 -21079.862} C_VEL
LIN {X 0,Y 206.753,Z 294.535,A -85,B 0,C 180,E1 -21084.066,E2 -21084.066} C_VEL
LIN {X 0,Y 206.724,Z 294.54,A -85,B 0,C 180,E1 -21088.413,E2 -21088.413} C_VEL
LIN {X 0,Y 206.678,Z 294.553,A -85,B 0,C 180,E1 -21093.535,E2 -21093.535} C_VEL
LIN {X 0,Y 206.732,Z 294.675,A -85,B 0,C 180,E1 -21093.891,E2 -21093.891} C_VEL
LIN {X 0,Y 207.69,Z 297.366,A -85,B 0,C 180,E1 -21094.298,E2 -21094.298} C_VEL
LIN {X 0,Y 209.795,Z 299.765,A -85,B 0,C 180,E1 -21094.998,E2 -21094.998} C_VEL
LIN {X 0,Y 211.984,Z 303.226,A -85,B 0,C 180,E1 -21095.747,E2 -21095.747} C_VEL
LIN {X 0,Y 213.669,Z 305.627,A -85,B 0,C 180,E1 -21096.294,E2 -21096.294} C_VEL
LIN {X 0,Y 218.344,Z 312.705,A -85,B 0,C 180,E1 -21097.767,E2 -21097.767} C_VEL
LIN {X 0,Y 224.75,Z 323.392,A -85,B 0,C 180,E1 -21099.678,E2 -21099.678} C_VEL
LIN {X 0,Y 228.652,Z 330.896,A -85,B 0,C 180,E1 -21100.804,E2 -21100.804} C_VEL
LIN {X 0,Y 230.924,Z 336.078,A -85,B 0,C 180,E1 -21101.459,E2 -21101.459} C_VEL
